C03649=1163.496,44.523,-49.145,-179.678,6.140,149.011
C03650=1163.500,44.274,-49.130,-179.680,6.139,149.011
C03651=1163.506,44.024,-49.115,-179.683,6.138,149.012
C03652=1163.511,43.775,-49.100,-179.686,6.137,149.012
C03653=1163.515,43.525,-49.084,-179.688,6.136,149.013
C03654=1163.521,43.275,-49.069,-179.691,6.135,149.014
C03655=1163.525,43.026,-49.054,-179.694,6.134,149.014
C03656=1163.531,42.777,-49.038,-179.696,6.133,149.015
C03657=1163.536,42.528,-49.023,-179.699,6.132,149.015
C03658=1163.540,42.278,-49.007,-179.701,6.131,149.016
C03659=1163.546,42.028,-48.992,-179.704,6.131,149.016
C03660=1163.551,41.779,-48.976,-179.707,6.129,149.017
C03661=1163.556,41.530,-48.961,-179.709,6.129,149.018
C03662=1163.561,41.280,-48.946,-179.711,6.128,149.018
C03663=1163.565,41.031,-48.930,-179.715,6.127,149.019
C03664=1163.571,40.781,-48.915,-179.717,6.126,149.019
C03665=1163.576,40.531,-48.900,-179.719,6.125,149.020
C03666=1163.581,40.282,-48.885,-179.722,6.124,149.020
C03667=1163.586,40.033,-48.869,-179.725,6.123,149.021
C03668=1163.591,39.784,-48.854,-179.727,6.122,149.021
C03669=1163.596,39.534,-48.839,-179.730,6.121,149.022
C03670=1163.601,39.284,-48.824,-179.732,6.120,149.022
C03671=1163.606,39.034,-48.808,-179.735,6.120,149.023
C03672=1163.611,38.785,-48.793,-179.737,6.119,149.024
C03673=1163.616,38.536,-48.778,-179.740,6.117,149.024
C03674=1163.621,38.286,-48.764,-179.742,6.117,149.025
C03675=1163.626,38.037,-48.748,-179.745,6.116,149.025
C03676=1163.632,37.787,-48.732,-179.748,6.114,149.026
C03677=1163.636,37.538,-48.717,-179.751,6.114,149.026
C03678=1163.642,37.288,-48.702,-179.753,6.113,149.027
C03679=1163.646,37.039,-48.687,-179.756,6.112,149.028
C03680=1163.652,36.789,-48.672,-179.758,6.111,149.028
C03681=1163.656,36.540,-48.657,-179.761,6.110,149.029
C03682=1163.661,36.290,-48.642,-179.763,6.110,149.029
C03683=1163.667,36.041,-48.627,-179.766,6.108,149.030
C03684=1163.671,35.792,-48.612,-179.768,6.107,149.030
C03685=1163.677,35.542,-48.597,-179.771,6.107,149.031
C03686=1163.682,35.293,-48.582,-179.774,6.105,149.031
C03687=1163.687,35.043,-48.566,-179.776,6.105,149.032
C03688=1163.692,34.794,-48.552,-179.779,6.104,149.033
C03689=1163.697,34.543,-48.536,-179.781,6.104,149.033
C03690=1163.702,34.294,-48.522,-179.784,6.102,149.034
C03691=1163.706,34.045,-48.507,-179.787,6.101,149.034
C03692=1163.712,33.795,-48.491,-179.789,6.101,149.035
C03693=1163.717,33.546,-48.477,-179.791,6.100,149.035
C03694=1163.722,33.296,-48.461,-179.795,6.099,149.036
C03695=1163.727,33.046,-48.447,-179.797,6.098,149.037
C03696=1163.732,32.797,-48.432,-179.799,6.097,149.037
C03697=1163.737,32.548,-48.416,-179.802,6.096,149.038
C03698=1163.742,32.298,-48.402,-179.805,6.095,149.038
C03699=1163.747,32.049,-48.387,-179.807,6.094,149.039
C03700=1163.752,31.799,-48.372,-179.810,6.094,149.040
C03701=1163.757,31.550,-48.357,-179.812,6.092,149.040
C03702=1163.763,31.300,-48.342,-179.815,6.092,149.041
C03703=1163.767,31.051,-48.327,-179.817,6.091,149.041
C03704=1163.772,30.801,-48.313,-179.820,6.091,149.042
C03705=1163.777,30.552,-48.298,-179.823,6.089,149.042
C03706=1163.783,30.302,-48.283,-179.825,6.088,149.043
C03707=1163.787,30.053,-48.268,-179.828,6.088,149.044
C03708=1163.792,29.803,-48.254,-179.830,6.087,149.044
C03709=1163.798,29.554,-48.238,-179.833,6.086,149.045
C03710=1163.803,29.304,-48.224,-179.835,6.085,149.045
C03711=1163.807,29.054,-48.210,-179.838,6.084,149.046
C03712=1163.813,28.805,-48.194,-179.840,6.084,149.046
C03713=1163.818,28.555,-48.180,-179.843,6.082,149.047
C03714=1163.823,28.287,-48.164,-179.846,6.082,149.048
C03715=1163.829,28.017,-48.148,-179.848,6.081,149.048
C03716=1163.834,27.749,-48.132,-179.851,6.080,149.049
C03717=1163.839,27.480,-48.117,-179.854,6.079,149.049
C03718=1163.844,27.230,-48.102,-179.856,6.078,149.050
C03719=1163.850,26.982,-48.087,-179.860,6.077,149.051
C03720=1163.855,26.732,-48.073,-179.862,6.076,149.051
C03721=1163.860,26.482,-48.059,-179.864,6.076,149.052
C03722=1163.865,26.233,-48.044,-179.866,6.075,149.052
C03723=1163.870,25.983,-48.029,-179.870,6.074,149.053
C03724=1163.875,25.733,-48.014,-179.872,6.073,149.054
C03725=1163.880,25.484,-47.999,-179.875,6.072,149.054
C03726=1163.885,25.234,-47.985,-179.877,6.072,149.055
C03727=1163.890,24.985,-47.971,-179.879,6.071,149.055
C03728=1163.895,24.735,-47.955,-179.883,6.070,149.056
C03729=1163.900,24.486,-47.941,-179.885,6.069,149.056
C03730=1163.905,24.236,-47.927,-179.887,6.069,149.057
C03731=1163.911,23.987,-47.913,-179.890,6.068,149.057
C03732=1163.915,23.738,-47.898,-179.893,6.066,149.058
C03733=1163.920,23.488,-47.884,-179.895,6.066,149.059
C03734=1163.925,23.238,-47.869,-179.898,6.065,149.059
C03735=1163.931,22.988,-47.854,-179.900,6.065,149.060
C03736=1163.936,22.739,-47.840,-179.902,6.064,149.060
C03737=1163.940,22.490,-47.825,-179.906,6.062,149.061
C03738=1163.945,22.240,-47.811,-179.908,6.062,149.061
C03739=1163.951,21.991,-47.797,-179.910,6.061,149.062
C03740=1163.956,21.741,-47.783,-179.913,6.060,149.063
C03741=1163.961,21.491,-47.768,-179.915,6.060,149.063
C03742=1163.966,21.242,-47.753,-179.918,6.058,149.064
C03743=1163.970,20.993,-47.739,-179.921,6.058,149.064
C03744=1163.976,20.743,-47.724,-179.923,6.057,149.065
C03745=1163.981,20.493,-47.710,-179.926,6.056,149.066
C03746=1163.987,20.244,-47.696,-179.928,6.056,149.066
C03747=1163.992,19.994,-47.682,-179.931,6.054,149.067
C03748=1163.997,19.744,-47.667,-179.934,6.054,149.067
C03749=1164.002,19.495,-47.653,-179.936,6.053,149.068
C03750=1164.006,19.246,-47.638,-179.938,6.053,149.069
C03751=1164.012,18.997,-47.624,-179.941,6.052,149.069
C03752=1164.017,18.747,-47.610,-179.943,6.051,149.070
C03753=1164.022,18.497,-47.596,-179.946,6.050,149.070
C03754=1164.027,18.248,-47.581,-179.949,6.049,149.071
C03755=1164.032,17.998,-47.567,-179.951,6.049,149.071
C03756=1164.037,17.749,-47.553,-179.953,6.048,149.072
C03757=1164.042,17.499,-47.539,-179.956,6.047,149.073
C03758=1164.047,17.249,-47.525,-179.959,6.046,149.073
C03759=1164.052,17.000,-47.510,-179.961,6.045,149.074
C03760=1164.057,16.750,-47.496,-179.964,6.044,149.074
C03761=1164.063,16.501,-47.482,-179.966,6.044,149.075
C03762=1164.067,16.251,-47.468,-179.968,6.043,149.075
C03763=1164.072,16.002,-47.454,-179.971,6.043,149.076
C03764=1164.077,15.752,-47.439,-179.974,6.041,149.077
C03765=1164.083,15.503,-47.426,-179.977,6.041,149.077
C03766=1164.088,15.253,-47.411,-179.979,6.040,149.078
C03767=1164.093,15.003,-47.397,-179.981,6.039,149.078
C03768=1164.098,14.754,-47.383,-179.984,6.039,149.079
C03769=1164.103,14.504,-47.370,-179.986,6.038,149.079
C03770=1164.108,14.255,-47.356,-179.989,6.037,149.080
C03771=1164.113,14.005,-47.342,-179.992,6.036,149.081
C03772=1164.118,13.756,-47.328,-179.994,6.035,149.081
C03773=1164.123,13.506,-47.313,-179.997,6.035,149.082
C03774=1164.128,13.257,-47.299,-179.999,6.034,149.082
C03775=1164.133,13.007,-47.285,179.998,6.034,149.083
C03776=1164.139,12.758,-47.271,179.996,6.033,149.084
C03777=1164.144,12.508,-47.257,179.993,6.032,149.084
C03778=1164.149,12.258,-47.243,179.991,6.031,149.085
C03779=1164.154,12.009,-47.230,179.988,6.030,149.085
C03780=1164.159,11.759,-47.215,179.985,6.030,149.086
C03781=1164.164,11.510,-47.201,179.983,6.029,149.087
C03782=1164.169,11.261,-47.187,179.981,6.028,149.087
C03783=1164.175,11.010,-47.174,179.978,6.028,149.088
C03784=1164.180,10.761,-47.159,179.976,6.027,149.088
C03785=1164.184,10.511,-47.146,179.973,6.026,149.089
C03786=1164.189,10.262,-47.132,179.970,6.025,149.089
C03787=1164.194,10.012,-47.118,179.968,6.025,149.090
C03788=1164.200,9.762,-47.104,179.966,6.024,149.091
C03789=1164.205,9.513,-47.090,179.963,6.023,149.091
C03790=1164.210,9.263,-47.076,179.961,6.022,149.092
C03791=1164.215,9.015,-47.062,179.958,6.022,149.092
C03792=1164.220,8.764,-47.049,179.956,6.021,149.093
C03793=1164.225,8.515,-47.035,179.953,6.020,149.094
C03794=1164.231,8.266,-47.021,179.950,6.019,149.094
C03795=1164.235,8.016,-47.008,179.948,6.019,149.095
C03796=1164.240,7.766,-46.993,179.945,6.018,149.095
C03797=1164.246,7.517,-46.980,179.943,6.017,149.096
C03798=1164.251,7.267,-46.966,179.940,6.017,149.097
C03799=1164.256,7.018,-46.953,179.938,6.016,149.097
C03800=1164.261,6.768,-46.938,179.936,6.016,149.098
C03801=1164.266,6.518,-46.925,179.933,6.014,149.098
C03802=1164.272,6.269,-46.911,179.930,6.013,149.099
C03803=1164.276,6.019,-46.897,179.927,6.013,149.100
C03804=1164.281,5.769,-46.884,179.925,6.012,149.100
C03805=1164.287,5.520,-46.870,179.923,6.012,149.101
C03806=1164.291,5.271,-46.856,179.920,6.011,149.101
C03807=1164.297,5.021,-46.843,179.918,6.010,149.102
C03808=1164.302,4.771,-46.829,179.916,6.010,149.102
C03809=1164.307,4.522,-46.815,179.913,6.009,149.103
C03810=1164.312,4.272,-46.802,179.910,6.009,149.104
C03811=1164.317,4.022,-46.788,179.908,6.007,149.104
C03812=1164.322,3.773,-46.774,179.905,6.007,149.105
C03813=1164.327,3.524,-46.761,179.903,6.006,149.105
C03814=1164.333,3.274,-46.747,179.900,6.005,149.106
C03815=1164.337,3.024,-46.733,179.898,6.005,149.106
C03816=1164.343,2.775,-46.721,179.895,6.004,149.107
C03817=1164.348,2.525,-46.706,179.893,6.004,149.108
C03818=1164.353,2.255,-46.692,179.890,6.003,149.108
C03819=1164.359,1.987,-46.678,179.887,6.002,149.109
C03820=1164.364,1.717,-46.663,179.885,6.001,149.110
C03821=1164.369,1.448,-46.648,179.882,6.001,149.110
C03822=1164.375,1.198,-46.635,179.880,6.000,149.111
C03823=1164.380,0.949,-46.621,179.877,5.999,149.112
C03824=1164.385,0.699,-46.608,179.875,5.998,149.112
C03825=1164.390,0.449,-46.595,179.872,5.998,149.113
C03826=1164.395,0.200,-46.581,179.870,5.998,149.113
C03827=1164.401,-0.050,-46.567,179.867,5.997,149.114
C03828=1164.406,-0.299,-46.554,179.864,5.996,149.115
C03829=1164.411,-0.549,-46.541,179.862,5.995,149.115
C03830=1164.416,-0.798,-46.528,179.859,5.994,149.116
C03831=1164.421,-1.048,-46.514,179.857,5.993,149.116
C03832=1164.426,-1.297,-46.501,179.855,5.993,149.117
C03833=1164.431,-1.547,-46.487,179.852,5.993,149.117
C03834=1164.436,-1.796,-46.474,179.850,5.992,149.118
C03835=1164.441,-2.047,-46.461,179.847,5.991,149.119
C03836=1164.446,-2.295,-46.447,179.845,5.990,149.119
C03837=1164.451,-2.546,-46.434,179.842,5.990,149.120
C03838=1164.457,-2.795,-46.421,179.840,5.989,149.120
C03839=1164.462,-3.045,-46.407,179.837,5.989,149.121
C03840=1164.467,-3.294,-46.394,179.835,5.988,149.122
C03841=1164.472,-3.544,-46.381,179.833,5.987,149.122
C03842=1164.477,-3.793,-46.367,179.830,5.987,149.123
C03843=1164.483,-4.043,-46.354,179.828,5.986,149.123
C03844=1164.487,-4.293,-46.341,179.825,5.986,149.124
C03845=1164.493,-4.542,-46.328,179.822,5.984,149.125
C03846=1164.497,-4.792,-46.314,179.820,5.984,149.125
C03847=1164.503,-5.041,-46.301,179.817,5.983,149.126
C03848=1164.508,-5.292,-46.288,179.815,5.982,149.126
C03849=1164.513,-5.541,-46.275,179.812,5.982,149.127
C03850=1164.518,-5.790,-46.262,179.810,5.981,149.127
C03851=1164.524,-6.040,-46.248,179.807,5.981,149.128
C03852=1164.529,-6.289,-46.236,179.805,5.980,149.129
C03853=1164.533,-6.539,-46.223,179.802,5.979,149.129
C03854=1164.539,-6.789,-46.209,179.800,5.979,149.130
C03855=1164.544,-7.038,-46.196,179.798,5.978,149.130
C03856=1164.549,-7.288,-46.183,179.795,5.978,149.131
C03857=1164.554,-7.537,-46.170,179.793,5.977,149.132
C03858=1164.559,-7.787,-46.157,179.790,5.976,149.132
C03859=1164.565,-8.037,-46.144,179.788,5.976,149.133
C03860=1164.569,-8.286,-46.130,179.785,5.975,149.133
C03861=1164.575,-8.536,-46.117,179.783,5.975,149.134
C03862=1164.580,-8.785,-46.104,179.780,5.974,149.135
C03863=1164.585,-9.035,-46.092,179.778,5.973,149.135
C03864=1164.590,-9.285,-46.078,179.776,5.973,149.136
C03865=1164.595,-9.534,-46.065,179.773,5.972,149.136
C03866=1164.600,-9.784,-46.053,179.770,5.972,149.137
C03867=1164.606,-10.034,-46.039,179.768,5.971,149.138
C03868=1164.611,-10.283,-46.026,179.766,5.970,149.138
C03869=1164.615,-10.533,-46.013,179.763,5.970,149.139
C03870=1164.621,-10.782,-46.000,179.761,5.969,149.139
C03871=1164.626,-11.032,-45.987,179.758,5.969,149.140
C03872=1164.631,-11.282,-45.974,179.756,5.968,149.141
C03873=1164.636,-11.531,-45.961,179.753,5.967,149.141
C03874=1164.642,-11.781,-45.948,179.751,5.967,149.142
C03875=1164.646,-12.031,-45.936,179.748,5.966,149.142
C03876=1164.651,-12.280,-45.923,179.746,5.965,149.143
C03877=1164.657,-12.530,-45.910,179.744,5.965,149.144
C03878=1164.662,-12.779,-45.897,179.741,5.964,149.144
C03879=1164.667,-13.029,-45.884,179.739,5.964,149.145
C03880=1164.673,-13.279,-45.871,179.736,5.963,149.145
C03881=1164.678,-13.528,-45.858,179.734,5.962,149.146
C03882=1164.682,-13.778,-45.845,179.731,5.962,149.147
C03883=1164.687,-14.027,-45.833,179.729,5.961,149.147
C03884=1164.693,-14.277,-45.820,179.726,5.961,149.148
C03885=1164.698,-14.527,-45.807,179.724,5.960,149.148
C03886=1164.703,-14.776,-45.794,179.722,5.959,149.149
C03887=1164.708,-15.026,-45.781,179.719,5.959,149.150
C03888=1164.713,-15.275,-45.769,179.717,5.958,149.150
C03889=1164.719,-15.526,-45.756,179.714,5.958,149.151
C03890=1164.724,-15.775,-45.743,179.711,5.957,149.151
C03891=1164.729,-16.024,-45.731,179.709,5.956,149.152
C03892=1164.734,-16.274,-45.718,179.707,5.956,149.153
C03893=1164.739,-16.524,-45.705,179.704,5.955,149.153
C03894=1164.744,-16.773,-45.692,179.702,5.955,149.154
C03895=1164.750,-17.023,-45.679,179.700,5.954,149.154
C03896=1164.755,-17.272,-45.667,179.697,5.953,149.155
C03897=1164.759,-17.523,-45.655,179.694,5.953,149.156
C03898=1164.765,-17.772,-45.642,179.692,5.952,149.156
C03899=1164.770,-18.021,-45.629,179.689,5.952,149.157
C03900=1164.776,-18.271,-45.616,179.687,5.951,149.157
C03901=1164.781,-18.520,-45.604,179.685,5.951,149.158
C03902=1164.785,-18.770,-45.591,179.682,5.950,149.158
C03903=1164.791,-19.020,-45.579,179.680,5.949,149.159
C03904=1164.796,-19.270,-45.566,179.677,5.949,149.160
C03905=1164.801,-19.519,-45.554,179.675,5.948,149.160
C03906=1164.806,-19.768,-45.541,179.672,5.948,149.161
C03907=1164.811,-20.019,-45.527,179.670,5.947,149.161
C03908=1164.817,-20.268,-45.515,179.667,5.946,149.162
C03909=1164.822,-20.518,-45.503,179.665,5.946,149.163
C03910=1164.827,-20.767,-45.490,179.663,5.946,149.163
C03911=1164.832,-21.017,-45.478,179.660,5.945,149.164
C03912=1164.838,-21.266,-45.466,179.658,5.945,149.165
C03913=1164.842,-21.516,-45.453,179.656,5.944,149.165
C03914=1164.847,-21.766,-45.440,179.653,5.943,149.166
C03915=1164.853,-22.016,-45.428,179.651,5.943,149.166
C03916=1164.858,-22.265,-45.416,179.648,5.943,149.167
C03917=1164.863,-22.514,-45.403,179.646,5.942,149.168
C03918=1164.868,-22.764,-45.391,179.643,5.941,149.168
C03919=1164.874,-23.015,-45.378,179.641,5.940,149.169
C03920=1164.879,-23.264,-45.365,179.638,5.940,149.169
C03921=1164.884,-23.514,-45.353,179.636,5.939,149.170
C03922=1164.890,-23.783,-45.340,179.634,5.939,149.171
C03923=1164.895,-24.053,-45.327,179.631,5.938,149.171
C03924=1164.901,-24.323,-45.313,179.628,5.938,149.172
C03925=1164.906,-24.592,-45.299,179.626,5.937,149.173
C03926=1164.911,-24.843,-45.287,179.623,5.937,149.173
C03927=1164.916,-25.092,-45.274,179.621,5.936,149.174
C03928=1164.922,-25.342,-45.263,179.619,5.935,149.174
C03929=1164.927,-25.591,-45.250,179.616,5.935,149.175
C03930=1164.932,-25.841,-45.237,179.614,5.934,149.175
C03931=1164.937,-26.091,-45.226,179.611,5.934,149.176
C03932=1164.943,-26.340,-45.213,179.608,5.933,149.177
C03933=1164.948,-26.590,-45.201,179.606,5.932,149.177
C03934=1164.953,-26.839,-45.188,179.604,5.932,149.178
C03935=1164.959,-27.089,-45.177,179.601,5.931,149.178
C03936=1164.962,-27.339,-45.164,179.599,5.932,149.179
C03937=1164.968,-27.589,-45.152,179.597,5.931,149.180
C03938=1164.973,-27.838,-45.140,179.594,5.930,149.180
C03939=1164.978,-28.088,-45.128,179.592,5.930,149.181
C03940=1164.983,-28.337,-45.115,179.590,5.929,149.182
C03941=1164.989,-28.587,-45.103,179.587,5.929,149.182
C03942=1164.994,-28.837,-45.091,179.585,5.928,149.183
C03943=1164.999,-29.087,-45.079,179.582,5.927,149.183
C03944=1165.005,-29.336,-45.066,179.580,5.927,149.184
C03945=1165.010,-29.586,-45.054,179.577,5.926,149.185
C03946=1165.015,-29.835,-45.042,179.575,5.926,149.185
C03947=1165.020,-30.085,-45.030,179.572,5.925,149.186
C03948=1165.025,-30.334,-45.018,179.570,5.925,149.186
C03949=1165.030,-30.584,-45.006,179.568,5.925,149.187
C03950=1165.035,-30.833,-44.993,179.566,5.924,149.188
C03951=1165.041,-31.083,-44.981,179.563,5.923,149.188
C03952=1165.046,-31.333,-44.970,179.561,5.923,149.189
C03953=1165.051,-31.583,-44.957,179.558,5.922,149.189
C03954=1165.056,-31.832,-44.946,179.556,5.922,149.190
C03955=1165.061,-32.082,-44.933,179.553,5.921,149.191
C03956=1165.067,-32.331,-44.921,179.551,5.920,149.191
C03957=1165.072,-32.581,-44.909,179.549,5.921,149.192
C03958=1165.077,-32.831,-44.897,179.547,5.920,149.192
C03959=1165.083,-33.081,-44.885,179.544,5.920,149.193
C03960=1165.087,-33.330,-44.874,179.541,5.919,149.194
C03961=1165.092,-33.580,-44.861,179.539,5.918,149.194
C03962=1165.098,-33.830,-44.849,179.537,5.918,149.195
C03963=1165.103,-34.079,-44.837,179.534,5.917,149.195
C03964=1165.108,-34.329,-44.825,179.532,5.917,149.196
C03965=1165.113,-34.578,-44.813,179.530,5.916,149.196
C03966=1165.119,-34.828,-44.801,179.528,5.916,149.197
C03967=1165.124,-35.078,-44.789,179.525,5.916,149.198
C03968=1165.129,-35.328,-44.777,179.523,5.915,149.198
C03969=1165.135,-35.578,-44.765,179.520,5.915,149.199
C03970=1165.139,-35.827,-44.754,179.518,5.914,149.200
C03971=1165.144,-36.076,-44.741,179.515,5.913,149.200
C03972=1165.150,-36.326,-44.729,179.513,5.913,149.201
C03973=1165.155,-36.576,-44.717,179.510,5.912,149.201
C03974=1165.160,-36.826,-44.706,179.509,5.912,149.202
C03975=1165.165,-37.075,-44.693,179.506,5.912,149.203
C03976=1165.170,-37.325,-44.682,179.503,5.911,149.203
C03977=1165.175,-37.575,-44.670,179.501,5.910,149.204
C03978=1165.181,-37.825,-44.658,179.499,5.910,149.204
C03979=1165.186,-38.073,-44.646,179.496,5.909,149.205
C03980=1165.192,-38.323,-44.634,179.494,5.909,149.206
C03981=1165.196,-38.573,-44.623,179.492,5.908,149.206
C03982=1165.202,-38.823,-44.611,179.489,5.908,149.207
C03983=1165.207,-39.073,-44.599,179.487,5.908,149.208
C03984=1165.212,-39.322,-44.588,179.485,5.907,149.208
C03985=1165.217,-39.572,-44.575,179.482,5.907,149.209
C03986=1165.223,-39.822,-44.563,179.480,5.906,149.209
C03987=1165.227,-40.071,-44.552,179.477,5.905,149.210
C03988=1165.233,-40.321,-44.540,179.475,5.905,149.210
C03989=1165.239,-40.571,-44.529,179.473,5.905,149.211
C03990=1165.243,-40.820,-44.517,179.471,5.904,149.211
C03991=1165.249,-41.070,-44.506,179.468,5.904,149.212
C03992=1165.254,-41.320,-44.494,179.465,5.903,149.213
C03993=1165.259,-41.569,-44.482,179.463,5.903,149.213
C03994=1165.264,-41.819,-44.470,179.460,5.902,149.214
C03995=1165.269,-42.069,-44.458,179.459,5.902,149.215
C03996=1165.274,-42.319,-44.447,179.456,5.902,149.215
C03997=1165.280,-42.568,-44.435,179.454,5.901,149.216
C03998=1165.285,-42.817,-44.424,179.451,5.901,149.216
C03999=1165.290,-43.067,-44.412,179.449,5.900,149.217
C04000=1165.296,-43.317,-44.400,179.447,5.899,149.218
C04001=1165.300,-43.567,-44.389,179.444,5.899,149.218
C04002=1165.306,-43.817,-44.377,179.442,5.899,149.219
C04003=1165.311,-44.066,-44.366,179.440,5.898,149.219
C04004=1165.317,-44.316,-44.354,179.437,5.898,149.220
C04005=1165.321,-44.565,-44.343,179.435,5.897,149.221
C04006=1165.327,-44.815,-44.331,179.433,5.896,149.221
C04007=1165.332,-45.065,-44.319,179.430,5.896,149.222
C04008=1165.337,-45.315,-44.308,179.428,5.896,149.222
C04009=1165.343,-45.564,-44.296,179.426,5.896,149.223
C04010=1165.348,-45.814,-44.285,179.423,5.895,149.224
C04011=1165.353,-46.064,-44.273,179.421,5.894,149.224
C04012=1165.358,-46.313,-44.262,179.418,5.894,149.225
C04013=1165.363,-46.563,-44.250,179.417,5.894,149.225
C04014=1165.368,-46.812,-44.239,179.414,5.894,149.226
C04015=1165.374,-47.062,-44.227,179.412,5.893,149.227
C04016=1165.379,-47.312,-44.216,179.409,5.892,149.227
C04017=1165.384,-47.562,-44.204,179.407,5.892,149.228
C04018=1165.389,-47.812,-44.193,179.404,5.891,149.228
C04019=1165.395,-48.061,-44.182,179.402,5.892,149.229
C04020=1165.400,-48.311,-44.170,179.400,5.891,149.230
C04021=1165.405,-48.561,-44.159,179.397,5.890,149.230
C04022=1165.410,-48.810,-44.147,179.395,5.889,149.231
C04023=1165.416,-49.059,-44.136,179.392,5.889,149.231
C04024=1165.421,-49.309,-44.125,179.391,5.889,149.232
C04025=1165.426,-49.559,-44.113,179.388,5.889,149.233
C04026=1165.432,-49.829,-44.101,179.385,5.888,149.233
C04027=1165.437,-50.100,-44.089,179.383,5.887,149.234
C04028=1165.442,-50.370,-44.076,179.381,5.887,149.235
C04029=1165.449,-50.641,-44.064,179.378,5.887,149.235
C04030=1165.454,-50.891,-44.052,179.376,5.886,149.236
C04031=1165.459,-51.141,-44.042,179.373,5.885,149.236
C04032=1165.464,-51.390,-44.030,179.371,5.885,149.237
C04033=1165.470,-51.640,-44.019,179.369,5.885,149.238
C04034=1165.474,-51.889,-44.008,179.366,5.885,149.238
C04035=1165.480,-52.139,-43.996,179.364,5.884,149.239
C04036=1165.485,-52.389,-43.986,179.361,5.883,149.240
C04037=1165.490,-52.638,-43.974,179.360,5.883,149.240
C04038=1165.496,-52.888,-43.962,179.357,5.883,149.241
C04039=1165.500,-53.138,-43.951,179.355,5.882,149.241
C04040=1165.507,-53.388,-43.940,179.352,5.882,149.242
C04041=1165.511,-53.637,-43.929,179.350,5.881,149.242
C04042=1165.516,-53.887,-43.918,179.348,5.881,149.243
C04043=1165.522,-54.136,-43.906,179.346,5.881,149.244
C04044=1165.527,-54.387,-43.896,179.343,5.880,149.244
C04045=1165.532,-54.636,-43.884,179.340,5.880,149.245
C04046=1165.538,-54.885,-43.873,179.338,5.879,149.245
C04047=1165.543,-55.136,-43.862,179.336,5.879,149.246
C04048=1165.547,-55.385,-43.851,179.334,5.879,149.247
C04049=1165.553,-55.635,-43.839,179.331,5.878,149.247
C04050=1165.558,-55.885,-43.829,179.329,5.877,149.248
C04051=1165.563,-56.134,-43.818,179.327,5.878,149.248
C04052=1165.569,-56.384,-43.806,179.325,5.877,149.249
C04053=1165.574,-56.634,-43.795,179.322,5.877,149.250
C04054=1165.579,-56.883,-43.784,179.320,5.876,149.250
C04055=1165.584,-57.132,-43.773,179.317,5.875,149.251
C04056=1165.590,-57.383,-43.762,179.316,5.875,149.251
C04057=1165.595,-57.633,-43.751,179.313,5.875,149.252
C04058=1165.600,-57.882,-43.741,179.311,5.874,149.252
C04059=1165.606,-58.132,-43.729,179.308,5.874,149.253
C04060=1165.610,-58.382,-43.717,179.306,5.874,149.254
C04061=1165.616,-58.631,-43.707,179.304,5.873,149.254
C04062=1165.621,-58.881,-43.696,179.301,5.873,149.255
C04063=1165.627,-59.131,-43.685,179.299,5.872,149.256
C04064=1165.632,-59.380,-43.674,179.297,5.872,149.256
C04065=1165.637,-59.631,-43.663,179.295,5.872,149.257
C04066=1165.642,-59.880,-43.652,179.292,5.871,149.257
C04067=1165.647,-60.129,-43.641,179.290,5.870,149.258
C04068=1165.652,-60.380,-43.630,179.288,5.871,149.259
C04069=1165.658,-60.629,-43.619,179.286,5.870,149.259
C04070=1165.663,-60.879,-43.608,179.283,5.870,149.260
C04071=1165.668,-61.128,-43.597,179.281,5.869,149.260
C04072=1165.674,-61.378,-43.586,179.279,5.869,149.261
C04073=1165.679,-61.627,-43.575,179.277,5.868,149.261
C04074=1165.684,-61.878,-43.565,179.274,5.868,149.262
C04075=1165.689,-62.127,-43.553,179.272,5.867,149.263
C04076=1165.694,-62.377,-43.543,179.270,5.868,149.263
C04077=1165.699,-62.626,-43.532,179.267,5.867,149.264
C04078=1165.705,-62.876,-43.521,179.265,5.866,149.265
C04079=1165.710,-63.126,-43.511,179.263,5.866,149.265
C04080=1165.716,-63.375,-43.500,179.261,5.866,149.266
C04081=1165.721,-63.626,-43.489,179.258,5.865,149.266
C04082=1165.725,-63.875,-43.478,179.256,5.865,149.267
C04083=1165.731,-64.125,-43.468,179.253,5.864,149.268
C04084=1165.736,-64.375,-43.456,179.251,5.864,149.268
C04085=1165.742,-64.624,-43.446,179.249,5.864,149.269
C04086=1165.747,-64.874,-43.435,179.247,5.863,149.269
C04087=1165.752,-65.123,-43.424,179.244,5.863,149.270
C04088=1165.757,-65.374,-43.413,179.242,5.863,149.270
C04089=1165.762,-65.623,-43.403,179.240,5.863,149.271
C04090=1165.767,-65.873,-43.392,179.237,5.862,149.272
C04091=1165.773,-66.122,-43.382,179.235,5.862,149.272
C04092=1165.778,-66.372,-43.370,179.233,5.861,149.273
C04093=1165.784,-66.622,-43.360,179.231,5.861,149.274
C04094=1165.789,-66.872,-43.349,179.228,5.860,149.274
C04095=1165.794,-67.121,-43.338,179.226,5.861,149.275
C04096=1165.799,-67.371,-43.328,179.224,5.860,149.275
C04097=1165.805,-67.621,-43.317,179.221,5.859,149.276
C04098=1165.810,-67.870,-43.306,179.219,5.859,149.276
C04099=1165.815,-68.120,-43.296,179.217,5.859,149.277
C04100=1165.820,-68.370,-43.285,179.215,5.858,149.278
C04101=1165.826,-68.619,-43.274,179.212,5.858,149.278
C04102=1165.831,-68.869,-43.264,179.211,5.858,149.279
C04103=1165.836,-69.119,-43.254,179.208,5.857,149.279
C04104=1165.841,-69.369,-43.243,179.206,5.857,149.280
C04105=1165.846,-69.618,-43.232,179.203,5.856,149.281
C04106=1165.851,-69.868,-43.222,179.202,5.856,149.281
C04107=1165.857,-70.118,-43.211,179.199,5.856,149.282
C04108=1165.863,-70.368,-43.200,179.197,5.855,149.282
C04109=1165.868,-70.617,-43.189,179.195,5.855,149.283
C04110=1165.873,-70.868,-43.179,179.192,5.855,149.284
C04111=1165.879,-71.117,-43.168,179.190,5.854,149.284
C04112=1165.884,-71.367,-43.158,179.188,5.853,149.285
C04113=1165.889,-71.616,-43.147,179.186,5.854,149.285
C04114=1165.895,-71.866,-43.137,179.183,5.853,149.286
C04115=1165.900,-72.116,-43.126,179.181,5.853,149.287
C04116=1165.905,-72.366,-43.116,179.179,5.853,149.287
C04117=1165.910,-72.616,-43.105,179.176,5.852,149.288
C04118=1165.916,-72.865,-43.095,179.174,5.851,149.288
C04119=1165.920,-73.114,-43.085,179.172,5.852,149.289
C04120=1165.925,-73.364,-43.074,179.170,5.851,149.289
C04121=1165.931,-73.614,-43.064,179.167,5.851,149.290
C04122=1165.936,-73.864,-43.053,179.165,5.850,149.291
C04123=1165.941,-74.114,-43.043,179.163,5.850,149.291
C04124=1165.947,-74.363,-43.033,179.161,5.849,149.292
C04125=1165.952,-74.613,-43.022,179.158,5.849,149.293
C04126=1165.957,-74.862,-43.012,179.157,5.849,149.293
C04127=1165.962,-75.113,-43.001,179.154,5.849,149.294
C04128=1165.968,-75.362,-42.991,179.152,5.848,149.294
C04129=1165.974,-75.612,-42.981,179.150,5.848,149.295
C04130=1165.979,-75.883,-42.970,179.147,5.848,149.295
C04131=1165.985,-76.155,-42.958,179.145,5.847,149.296
C04132=1165.991,-76.425,-42.947,179.142,5.847,149.297
C04133=1165.996,-76.697,-42.936,179.140,5.846,149.297
C04134=1166.002,-76.946,-42.926,179.138,5.846,149.298
C04135=1166.007,-77.197,-42.915,179.136,5.846,149.299
C04136=1166.013,-77.446,-42.905,179.133,5.845,149.299
C04137=1166.018,-77.696,-42.895,179.131,5.845,149.300
C04138=1166.023,-77.945,-42.883,179.129,5.845,149.300
C04139=1166.028,-78.194,-42.874,179.126,5.844,149.301
C04140=1166.033,-78.444,-42.864,179.124,5.844,149.302
C04141=1166.038,-78.694,-42.853,179.122,5.844,149.302
C04142=1166.044,-78.944,-42.843,179.120,5.843,149.303
C04143=1166.050,-79.193,-42.833,179.118,5.843,149.303
C04144=1166.055,-79.444,-42.822,179.115,5.843,149.304
C04145=1166.059,-79.693,-42.812,179.113,5.842,149.304
C04146=1166.065,-79.943,-42.803,179.111,5.842,149.305
C04147=1166.070,-80.193,-42.792,179.109,5.842,149.306
C04148=1166.076,-80.443,-42.782,179.107,5.841,149.306
C04149=1166.081,-80.692,-42.772,179.105,5.841,149.307
C04150=1166.086,-80.943,-42.761,179.102,5.841,149.307
C04151=1166.091,-81.192,-42.752,179.100,5.840,149.308
C04152=1166.097,-81.441,-42.742,179.098,5.840,149.309
C04153=1166.102,-81.692,-42.731,179.095,5.840,149.309
C04154=1166.108,-81.941,-42.721,179.093,5.839,149.310
C04155=1166.113,-82.191,-42.711,179.091,5.839,149.310
C04156=1166.117,-82.441,-42.701,179.089,5.839,149.311
C04157=1166.123,-82.690,-42.690,179.086,5.838,149.312
C04158=1166.129,-82.940,-42.680,179.085,5.838,149.312
C04159=1166.134,-83.190,-42.671,179.082,5.838,149.313
C04160=1166.139,-83.440,-42.661,179.080,5.837,149.313
C04161=1166.144,-83.689,-42.651,179.078,5.837,149.314
C04162=1166.150,-83.939,-42.640,179.076,5.837,149.314
C04163=1166.155,-84.189,-42.630,179.073,5.836,149.315
C04164=1166.160,-84.438,-42.620,179.071,5.836,149.316
C04165=1166.165,-84.688,-42.610,179.069,5.836,149.316
C04166=1166.171,-84.938,-42.600,179.066,5.835,149.317
C04167=1166.176,-85.188,-42.590,179.065,5.835,149.317
C04168=1166.181,-85.438,-42.580,179.062,5.835,149.318
C04169=1166.187,-85.687,-42.570,179.060,5.834,149.319
C04170=1166.192,-85.937,-42.560,179.058,5.834,149.319
C04171=1166.197,-86.187,-42.550,179.056,5.834,149.320
C04172=1166.203,-86.437,-42.540,179.054,5.834,149.320
C04173=1166.208,-86.686,-42.530,179.051,5.833,149.321
C04174=1166.213,-86.935,-42.521,179.049,5.832,149.321
C04175=1166.218,-87.186,-42.510,179.047,5.833,149.322
C04176=1166.224,-87.436,-42.500,179.045,5.832,149.323
C04177=1166.229,-87.685,-42.491,179.042,5.832,149.323
C04178=1166.234,-87.935,-42.481,179.041,5.832,149.324
C04179=1166.240,-88.184,-42.470,179.038,5.831,149.325
C04180=1166.245,-88.435,-42.461,179.036,5.831,149.325
C04181=1166.250,-88.684,-42.451,179.034,5.831,149.325
C04182=1166.256,-88.934,-42.441,179.032,5.830,149.326
C04183=1166.261,-89.183,-42.431,179.030,5.830,149.327
C04184=1166.266,-89.434,-42.421,179.027,5.830,149.327
C04185=1166.271,-89.683,-42.412,179.025,5.829,149.328
C04186=1166.276,-89.933,-42.401,179.023,5.829,149.329
C04187=1166.282,-90.183,-42.392,179.021,5.829,149.329
C04188=1166.287,-90.432,-42.382,179.019,5.828,149.330
C04189=1166.293,-90.682,-42.372,179.017,5.828,149.330
C04190=1166.298,-90.933,-42.362,179.014,5.828,149.331
C04191=1166.303,-91.182,-42.353,179.012,5.828,149.331
C04192=1166.308,-91.431,-42.342,179.010,5.827,149.332
C04193=1166.314,-91.681,-42.334,179.007,5.827,149.333
C04194=1166.319,-91.931,-42.323,179.006,5.827,149.333
C04195=1166.325,-92.180,-42.313,179.004,5.826,149.334
C04196=1166.329,-92.431,-42.304,179.001,5.826,149.334
C04197=1166.335,-92.680,-42.294,178.999,5.826,149.335
C04198=1166.340,-92.930,-42.284,178.997,5.825,149.336
C04199=1166.346,-93.180,-42.275,178.995,5.825,149.336
C04200=1166.351,-93.429,-42.265,178.992,5.825,149.337
C04201=1166.357,-93.679,-42.255,178.990,5.824,149.337
C04202=1166.361,-93.929,-42.245,178.989,5.824,149.338
C04203=1166.366,-94.179,-42.235,178.986,5.824,149.338
C04204=1166.372,-94.429,-42.226,178.984,5.824,149.339
C04205=1166.377,-94.678,-42.216,178.982,5.823,149.340
C04206=1166.383,-94.928,-42.207,178.979,5.823,149.340
C04207=1166.388,-95.177,-42.197,178.977,5.823,149.341
C04208=1166.394,-95.428,-42.188,178.975,5.822,149.341
C04209=1166.399,-95.677,-42.178,178.974,5.822,149.342
C04210=1166.404,-95.928,-42.168,178.971,5.822,149.342
C04211=1166.409,-96.177,-42.158,178.969,5.821,149.343
C04212=1166.414,-96.426,-42.148,178.967,5.822,149.344
C04213=1166.420,-96.676,-42.139,178.964,5.821,149.344
C04214=1166.425,-96.926,-42.129,178.963,5.821,149.345
C04215=1166.430,-97.176,-42.120,178.960,5.820,149.345
C04216=1166.436,-97.425,-42.110,178.958,5.820,149.346
C04217=1166.441,-97.675,-42.101,178.956,5.820,149.347
C04218=1166.447,-97.925,-42.092,178.954,5.819,149.347
C04219=1166.452,-98.174,-42.082,178.952,5.819,149.347
C04220=1166.458,-98.425,-42.073,178.949,5.819,149.348
C04221=1166.463,-98.674,-42.063,178.947,5.818,149.349
C04222=1166.468,-98.925,-42.053,178.945,5.819,149.349
C04223=1166.473,-99.174,-42.043,178.943,5.818,149.350
C04224=1166.478,-99.424,-42.035,178.941,5.818,149.350
C04225=1166.484,-99.673,-42.024,178.939,5.817,149.351
C04226=1166.489,-99.923,-42.015,178.937,5.817,149.352
C04227=1166.494,-100.173,-42.005,178.934,5.817,149.352
C04228=1166.500,-100.423,-41.996,178.932,5.816,149.353
C04229=1166.505,-100.673,-41.987,178.931,5.816,149.353
C04230=1166.510,-100.922,-41.977,178.928,5.816,149.354
C04231=1166.515,-101.172,-41.968,178.926,5.816,149.354
C04232=1166.521,-101.421,-41.958,178.924,5.816,149.355
C04233=1166.526,-101.671,-41.949,178.922,5.815,149.356
C04234=1166.532,-101.943,-41.939,178.919,5.815,149.356
C04235=1166.538,-102.215,-41.928,178.917,5.814,149.357
C04236=1166.543,-102.487,-41.918,178.915,5.814,149.358
C04237=1166.550,-102.759,-41.908,178.913,5.814,149.358
C04238=1166.555,-103.008,-41.899,178.910,5.814,149.359
C04239=1166.561,-103.259,-41.890,178.908,5.813,149.359
C04240=1166.565,-103.508,-41.880,178.906,5.813,149.360
C04241=1166.571,-103.758,-41.871,178.904,5.813,149.360
C04242=1166.577,-104.008,-41.862,178.902,5.813,149.361
C04243=1166.581,-104.257,-41.852,178.900,5.812,149.362
C04244=1166.587,-104.507,-41.843,178.898,5.812,149.362
C04245=1166.592,-104.757,-41.834,178.896,5.812,149.363
C04246=1166.597,-105.006,-41.824,178.893,5.811,149.363
C04247=1166.602,-105.256,-41.815,178.892,5.811,149.364
C04248=1166.608,-105.506,-41.806,178.889,5.811,149.365
C04249=1166.614,-105.756,-41.797,178.887,5.811,149.365
C04250=1166.618,-106.005,-41.787,178.885,5.810,149.366
C04251=1166.624,-106.256,-41.778,178.883,5.810,149.366
C04252=1166.629,-106.505,-41.769,178.881,5.810,149.367
C04253=1166.635,-106.755,-41.760,178.879,5.809,149.367
C04254=1166.640,-107.005,-41.750,178.877,5.809,149.368
C04255=1166.645,-107.255,-41.741,178.874,5.809,149.368
C04256=1166.651,-107.504,-41.732,178.873,5.809,149.369
C04257=1166.656,-107.754,-41.723,178.870,5.808,149.370
C04258=1166.661,-108.004,-41.713,178.868,5.808,149.370
C04259=1166.667,-108.254,-41.704,178.866,5.808,149.371
C04260=1166.672,-108.504,-41.695,178.864,5.808,149.371
C04261=1166.677,-108.753,-41.686,178.862,5.807,149.372
C04262=1166.683,-109.004,-41.677,178.859,5.807,149.372
C04263=1166.688,-109.253,-41.667,178.858,5.807,149.373
C04264=1166.693,-109.503,-41.658,178.855,5.806,149.373
C04265=1166.698,-109.753,-41.649,178.853,5.806,149.374
C04266=1166.704,-110.003,-41.640,178.851,5.806,149.375
C04267=1166.709,-110.253,-41.631,178.850,5.806,149.375
C04268=1166.714,-110.502,-41.622,178.847,5.805,149.376
C04269=1166.720,-110.751,-41.613,178.845,5.805,149.376
C04270=1166.726,-111.001,-41.603,178.843,5.805,149.377
C04271=1166.731,-111.251,-41.594,178.841,5.805,149.378
C04272=1166.736,-111.501,-41.585,178.839,5.804,149.378
C04273=1166.741,-111.751,-41.576,178.837,5.803,149.379
C04274=1166.746,-112.000,-41.568,178.835,5.804,149.379
C04275=1166.752,-112.251,-41.558,178.832,5.803,149.380
C04276=1166.757,-112.501,-41.549,178.830,5.804,149.380
C04277=1166.762,-112.750,-41.540,178.828,5.803,149.381
C04278=1166.767,-113.000,-41.531,178.827,5.803,149.381
C04279=1166.773,-113.249,-41.522,178.824,5.802,149.382
C04280=1166.779,-113.499,-41.513,178.822,5.802,149.383
C04281=1166.784,-113.749,-41.504,178.820,5.802,149.383
C04282=1166.789,-113.999,-41.495,178.818,5.802,149.384
C04283=1166.794,-114.248,-41.486,178.816,5.801,149.384
C04284=1166.800,-114.498,-41.477,178.814,5.801,149.385
C04285=1166.805,-114.748,-41.468,178.812,5.801,149.385
C04286=1166.811,-114.998,-41.459,178.810,5.801,149.386
C04287=1166.816,-115.247,-41.450,178.808,5.800,149.386
C04288=1166.822,-115.497,-41.441,178.806,5.800,149.387
C04289=1166.827,-115.747,-41.432,178.803,5.800,149.388
C04290=1166.832,-115.997,-41.423,178.801,5.799,149.388
C04291=1166.837,-116.247,-41.415,178.800,5.799,149.389
C04292=1166.842,-116.497,-41.406,178.797,5.799,149.389
C04293=1166.848,-116.747,-41.396,178.795,5.799,149.390
C04294=1166.854,-116.996,-41.388,178.793,5.798,149.390
C04295=1166.859,-117.246,-41.379,178.791,5.799,149.391
C04296=1166.864,-117.496,-41.370,178.789,5.798,149.392
C04297=1166.869,-117.746,-41.361,178.787,5.798,149.392
C04298=1166.875,-117.995,-41.352,178.785,5.797,149.393
C04299=1166.880,-118.245,-41.343,178.783,5.797,149.393
C04300=1166.886,-118.494,-41.335,178.781,5.797,149.394
C04301=1166.891,-118.744,-41.326,178.779,5.797,149.394
C04302=1166.896,-118.994,-41.317,178.777,5.796,149.395
C04303=1166.901,-119.244,-41.308,178.775,5.796,149.395
C04304=1166.906,-119.494,-41.299,178.772,5.796,149.396
C04305=1166.913,-119.744,-41.291,178.771,5.796,149.397
C04306=1166.918,-119.994,-41.282,178.769,5.795,149.397
C04307=1166.923,-120.244,-41.273,178.767,5.795,149.398
C04308=1166.929,-120.493,-41.264,178.764,5.795,149.398
C04309=1166.934,-120.743,-41.255,178.763,5.795,149.399
C04310=1166.939,-120.992,-41.246,178.760,5.794,149.399
C04311=1166.945,-121.242,-41.238,178.758,5.795,149.400
C04312=1166.950,-121.492,-41.229,178.756,5.794,149.400
C04313=1166.955,-121.742,-41.220,178.755,5.794,149.401
C04314=1166.960,-121.993,-41.212,178.752,5.793,149.401
C04315=1166.966,-122.242,-41.203,178.750,5.794,149.402
C04316=1166.971,-122.492,-41.194,178.748,5.793,149.403
C04317=1166.977,-122.741,-41.185,178.746,5.793,149.403
C04318=1166.982,-122.991,-41.176,178.744,5.792,149.404
C04319=1166.987,-123.240,-41.168,178.742,5.792,149.404
C04320=1166.993,-123.491,-41.160,178.740,5.792,149.405
C04321=1166.998,-123.741,-41.151,178.738,5.792,149.406
C04322=1167.003,-123.991,-41.142,178.736,5.791,149.406
C04323=1167.009,-124.240,-41.133,178.734,5.791,149.406
C04324=1167.014,-124.490,-41.124,178.732,5.791,149.407
C04325=1167.020,-124.740,-41.116,178.730,5.791,149.408
C04326=1167.025,-124.990,-41.107,178.728,5.790,149.408
C04327=1167.031,-125.239,-41.099,178.726,5.790,149.409
C04328=1167.036,-125.489,-41.090,178.724,5.790,149.409
C04329=1167.041,-125.739,-41.082,178.722,5.790,149.410
C04330=1167.046,-125.989,-41.073,178.720,5.789,149.410
C04331=1167.051,-126.238,-41.065,178.718,5.789,149.411
C04332=1167.057,-126.488,-41.056,178.715,5.789,149.412
C04333=1167.062,-126.738,-41.048,178.714,5.789,149.412
C04334=1167.068,-126.987,-41.039,178.712,5.788,149.413
C04335=1167.073,-127.237,-41.030,178.710,5.788,149.413
C04336=1167.078,-127.487,-41.021,178.707,5.788,149.414
C04337=1167.084,-127.738,-41.013,178.706,5.788,149.414
C04338=1166.663,-127.749,-41.054,178.702,5.791,149.416
C04339=1166.657,-127.498,-41.063,178.704,5.791,149.415
C04340=1166.652,-127.249,-41.072,178.706,5.791,149.415
C04341=1166.646,-126.999,-41.080,178.708,5.791,149.414
C04342=1166.641,-126.749,-41.088,178.710,5.792,149.414
C04343=1166.636,-126.499,-41.097,178.712,5.792,149.413
C04344=1166.631,-126.249,-41.106,178.714,5.793,149.413
C04345=1166.625,-126.000,-41.115,178.716,5.793,149.412
C04346=1166.619,-125.750,-41.123,178.718,5.793,149.412
C04347=1166.614,-125.500,-41.132,178.720,5.793,149.411
C04348=1166.609,-125.250,-41.141,178.722,5.794,149.410
C04349=1166.603,-125.001,-41.149,178.724,5.794,149.410
C04350=1166.598,-124.750,-41.157,178.726,5.794,149.410
C04351=1166.593,-124.500,-41.166,178.728,5.794,149.409
C04352=1166.587,-124.251,-41.175,178.730,5.795,149.408
C04353=1166.582,-124.001,-41.184,178.732,5.795,149.408
C04354=1166.577,-123.752,-41.192,178.735,5.795,149.407
C04355=1166.572,-123.501,-41.200,178.736,5.795,149.407
C04356=1166.566,-123.252,-41.209,178.738,5.796,149.406
C04357=1166.561,-123.002,-41.218,178.740,5.796,149.406
C04358=1166.556,-122.753,-41.226,178.743,5.796,149.405
C04359=1166.551,-122.503,-41.235,178.744,5.796,149.404
C04360=1166.545,-122.253,-41.244,178.746,5.797,149.404
C04361=1166.539,-122.003,-41.252,178.748,5.797,149.403
C04362=1166.534,-121.753,-41.261,178.751,5.797,149.403
C04363=1166.529,-121.503,-41.270,178.752,5.797,149.402
C04364=1166.523,-121.253,-41.279,178.754,5.798,149.402
C04365=1166.517,-121.004,-41.288,178.757,5.797,149.401
C04366=1166.512,-120.754,-41.297,178.759,5.798,149.401
C04367=1166.507,-120.504,-41.306,178.760,5.798,149.400
C04368=1166.502,-120.255,-41.315,178.763,5.799,149.399
C04369=1166.496,-120.004,-41.323,178.765,5.799,149.399
C04370=1166.491,-119.755,-41.331,178.767,5.799,149.398
C04371=1166.485,-119.505,-41.340,178.768,5.799,149.398
C04372=1166.480,-119.255,-41.349,178.771,5.800,149.397
C04373=1166.475,-119.005,-41.358,178.773,5.800,149.397
C04374=1166.470,-118.755,-41.367,178.775,5.800,149.396
C04375=1166.465,-118.506,-41.376,178.778,5.801,149.396
C04376=1166.459,-118.257,-41.384,178.779,5.801,149.395
C04377=1166.454,-118.007,-41.393,178.781,5.801,149.395
C04378=1166.449,-117.757,-41.402,178.783,5.801,149.394
C04379=1166.444,-117.507,-41.411,178.786,5.802,149.393
C04380=1166.438,-117.257,-41.420,178.787,5.802,149.393
C04381=1166.432,-117.008,-41.429,178.789,5.803,149.392
C04382=1166.427,-116.758,-41.438,178.792,5.802,149.392
C04383=1166.422,-116.508,-41.447,178.794,5.803,149.391
C04384=1166.416,-116.258,-41.456,178.795,5.803,149.391
C04385=1166.411,-116.008,-41.465,178.798,5.803,149.390
C04386=1166.406,-115.758,-41.473,178.800,5.803,149.389
C04387=1166.401,-115.509,-41.482,178.802,5.804,149.389
C04388=1166.395,-115.259,-41.491,178.804,5.804,149.388
C04389=1166.389,-115.009,-41.500,178.806,5.804,149.388
C04390=1166.384,-114.759,-41.509,178.808,5.804,149.387
C04391=1166.379,-114.510,-41.518,178.810,5.805,149.387
C04392=1166.374,-114.260,-41.527,178.812,5.805,149.386
C04393=1166.369,-114.010,-41.536,178.814,5.805,149.386
C04394=1166.363,-113.760,-41.545,178.816,5.805,149.385
C04395=1166.357,-113.510,-41.554,178.818,5.806,149.384
C04396=1166.352,-113.261,-41.563,178.821,5.806,149.384
C04397=1166.346,-113.011,-41.572,178.823,5.806,149.383
C04398=1166.341,-112.761,-41.581,178.825,5.807,149.383
C04399=1166.336,-112.511,-41.590,178.826,5.807,149.382
C04400=1166.331,-112.261,-41.599,178.829,5.807,149.382
C04401=1166.325,-112.011,-41.608,178.831,5.807,149.381
C04402=1166.320,-111.762,-41.618,178.833,5.808,149.381
C04403=1166.315,-111.512,-41.627,178.835,5.807,149.380
C04404=1166.309,-111.263,-41.635,178.837,5.808,149.379
C04405=1166.303,-111.013,-41.645,178.839,5.808,149.379
C04406=1166.298,-110.763,-41.653,178.841,5.809,149.378
C04407=1166.293,-110.513,-41.662,178.844,5.809,149.378
C04408=1166.288,-110.263,-41.671,178.845,5.809,149.377
C04409=1166.283,-110.013,-41.680,178.848,5.810,149.376
C04410=1166.277,-109.764,-41.690,178.850,5.810,149.376
C04411=1166.272,-109.514,-41.699,178.852,5.810,149.376
C04412=1166.267,-109.264,-41.708,178.854,5.810,149.375
C04413=1166.262,-109.014,-41.717,178.856,5.811,149.374
C04414=1166.256,-108.764,-41.727,178.858,5.811,149.374
C04415=1166.251,-108.515,-41.736,178.860,5.811,149.373
C04416=1166.246,-108.265,-41.745,178.862,5.811,149.373
C04417=1166.241,-108.015,-41.754,178.865,5.811,149.372
C04418=1166.235,-107.765,-41.763,178.867,5.812,149.371
C04419=1166.229,-107.516,-41.772,178.868,5.812,149.371
C04420=1166.224,-107.267,-41.782,178.871,5.813,149.370
C04421=1166.218,-107.016,-41.791,178.873,5.813,149.370
C04422=1166.213,-106.767,-41.800,178.875,5.813,149.369
C04423=1166.208,-106.517,-41.809,178.877,5.813,149.369
C04424=1166.203,-106.267,-41.818,178.879,5.814,149.368
C04425=1166.197,-106.017,-41.828,178.881,5.814,149.368
C04426=1166.192,-105.767,-41.837,178.883,5.814,149.367
C04427=1166.187,-105.518,-41.846,178.886,5.815,149.366
C04428=1166.181,-105.268,-41.856,178.888,5.814,149.366
C04429=1166.176,-105.018,-41.865,178.890,5.815,149.365
C04430=1166.171,-104.768,-41.874,178.891,5.815,149.365
C04431=1166.165,-104.518,-41.883,178.894,5.816,149.364
C04432=1166.160,-104.269,-41.893,178.896,5.815,149.363
C04433=1166.155,-104.019,-41.902,178.898,5.816,149.363
C04434=1166.149,-103.769,-41.911,178.901,5.817,149.362
C04435=1166.144,-103.520,-41.921,178.902,5.817,149.362
C04436=1166.139,-103.270,-41.930,178.905,5.817,149.361
C04437=1166.133,-103.020,-41.939,178.906,5.817,149.361
C04438=1166.128,-102.770,-41.949,178.909,5.818,149.360
C04439=1166.123,-102.499,-41.959,178.911,5.818,149.359
C04440=1166.117,-102.227,-41.969,178.913,5.818,149.359
C04441=1166.111,-101.954,-41.980,178.916,5.818,149.358
C04442=1166.105,-101.682,-41.990,178.918,5.819,149.357
C04443=1166.100,-101.433,-41.999,178.920,5.819,149.357
C04444=1166.094,-101.182,-42.009,178.922,5.820,149.357
C04445=1166.089,-100.933,-42.018,178.924,5.819,149.356
C04446=1166.084,-100.683,-42.027,178.926,5.820,149.355
C04447=1166.078,-100.433,-42.037,178.929,5.820,149.355
C04448=1166.074,-100.184,-42.046,178.931,5.820,149.354
C04449=1166.068,-99.934,-42.056,178.933,5.821,149.354
C04450=1166.063,-99.685,-42.066,178.935,5.821,149.353
C04451=1166.057,-99.434,-42.075,178.937,5.821,149.352
C04452=1166.052,-99.185,-42.085,178.940,5.822,149.352
C04453=1166.047,-98.935,-42.094,178.941,5.822,149.351
C04454=1166.041,-98.685,-42.103,178.944,5.823,149.351
C04455=1166.036,-98.436,-42.113,178.946,5.822,149.350
C04456=1166.030,-98.186,-42.122,178.948,5.823,149.350
C04457=1166.025,-97.937,-42.132,178.950,5.823,149.349
C04458=1166.019,-97.686,-42.141,178.952,5.823,149.348
C04459=1166.015,-97.436,-42.151,178.954,5.824,149.348
C04460=1166.009,-97.186,-42.161,178.956,5.824,149.347
C04461=1166.004,-96.937,-42.170,178.959,5.824,149.347
C04462=1165.998,-96.687,-42.180,178.961,5.825,149.346
C04463=1165.994,-96.438,-42.189,178.963,5.825,149.345
C04464=1165.988,-96.187,-42.199,178.965,5.826,149.345
C04465=1165.983,-95.938,-42.209,178.967,5.825,149.344
C04466=1165.977,-95.688,-42.218,178.969,5.826,149.344
C04467=1165.972,-95.439,-42.228,178.972,5.826,149.343
C04468=1165.966,-95.189,-42.237,178.974,5.826,149.343
C04469=1165.962,-94.939,-42.247,178.976,5.827,149.342
C04470=1165.956,-94.689,-42.257,178.978,5.827,149.341
C04471=1165.951,-94.439,-42.266,178.980,5.827,149.341
C04472=1165.946,-94.190,-42.276,178.983,5.828,149.340
C04473=1165.940,-93.940,-42.285,178.984,5.828,149.340
C04474=1165.935,-93.690,-42.296,178.986,5.829,149.339
C04475=1165.929,-93.440,-42.305,178.989,5.828,149.339
C04476=1165.924,-93.191,-42.315,178.991,5.829,149.338
C04477=1165.919,-92.941,-42.325,178.993,5.829,149.337
C04478=1165.914,-92.691,-42.334,178.995,5.829,149.337
C04479=1165.908,-92.441,-42.344,178.998,5.830,149.336
C04480=1165.903,-92.192,-42.353,178.999,5.830,149.336
C04481=1165.898,-91.942,-42.363,179.001,5.830,149.335
C04482=1165.892,-91.692,-42.374,179.004,5.831,149.334
C04483=1165.887,-91.442,-42.383,179.006,5.831,149.334
C04484=1165.882,-91.192,-42.393,179.008,5.831,149.333
C04485=1165.877,-90.943,-42.403,179.011,5.832,149.333
C04486=1165.871,-90.693,-42.412,179.013,5.832,149.332
C04487=1165.865,-90.443,-42.422,179.015,5.832,149.332
C04488=1165.861,-90.194,-42.432,179.016,5.832,149.331
C04489=1165.855,-89.943,-42.442,179.019,5.833,149.330
C04490=1165.850,-89.694,-42.451,179.021,5.833,149.330
C04491=1165.845,-89.445,-42.462,179.023,5.833,149.329
C04492=1165.839,-89.194,-42.471,179.026,5.834,149.329
C04493=1165.834,-88.945,-42.481,179.028,5.834,149.328
C04494=1165.829,-88.695,-42.491,179.030,5.834,149.328
C04495=1165.823,-88.445,-42.502,179.032,5.835,149.327
C04496=1165.818,-88.196,-42.510,179.034,5.835,149.326
C04497=1165.813,-87.946,-42.521,179.036,5.835,149.326
C04498=1165.808,-87.696,-42.531,179.039,5.836,149.325
C04499=1165.803,-87.446,-42.541,179.041,5.836,149.325
C04500=1165.797,-87.196,-42.550,179.043,5.836,149.324
C04501=1165.791,-86.947,-42.561,179.045,5.837,149.323
C04502=1165.786,-86.698,-42.570,179.048,5.836,149.323
C04503=1165.781,-86.447,-42.581,179.050,5.837,149.322
C04504=1165.776,-86.197,-42.590,179.052,5.838,149.322
C04505=1165.771,-85.948,-42.600,179.054,5.838,149.321
C04506=1165.765,-85.698,-42.610,179.056,5.838,149.321
C04507=1165.760,-85.448,-42.621,179.059,5.839,149.320
C04508=1165.755,-85.199,-42.630,179.060,5.839,149.319
C04509=1165.750,-84.949,-42.640,179.063,5.839,149.319
C04510=1165.744,-84.699,-42.650,179.065,5.839,149.318
C04511=1165.739,-84.449,-42.661,179.067,5.840,149.318
C04512=1165.734,-84.200,-42.670,179.070,5.840,149.317
C04513=1165.728,-83.950,-42.680,179.071,5.840,149.317
C04514=1165.723,-83.700,-42.691,179.074,5.841,149.316
C04515=1165.718,-83.451,-42.701,179.076,5.841,149.315
C04516=1165.712,-83.201,-42.710,179.078,5.841,149.315
C04517=1165.707,-82.951,-42.720,179.080,5.842,149.314
C04518=1165.702,-82.701,-42.731,179.083,5.842,149.313
C04519=1165.697,-82.452,-42.740,179.085,5.842,149.313
C04520=1165.691,-82.202,-42.751,179.087,5.843,149.312
C04521=1165.686,-81.952,-42.761,179.089,5.843,149.312
C04522=1165.681,-81.702,-42.771,179.092,5.843,149.311
C04523=1165.675,-81.453,-42.782,179.094,5.844,149.311
C04524=1165.670,-81.203,-42.791,179.096,5.845,149.310
C04525=1165.665,-80.953,-42.802,179.098,5.844,149.309
C04526=1165.660,-80.704,-42.812,179.100,5.845,149.309
C04527=1165.654,-80.454,-42.822,179.103,5.845,149.308
C04528=1165.649,-80.203,-42.832,179.104,5.845,149.308
C04529=1165.644,-79.954,-42.842,179.107,5.846,149.307
C04530=1165.638,-79.704,-42.852,179.109,5.846,149.307
C04531=1165.633,-79.454,-42.863,179.111,5.846,149.306
C04532=1165.628,-79.205,-42.873,179.114,5.847,149.305
C04533=1165.622,-78.955,-42.883,179.116,5.847,149.305
C04534=1165.617,-78.705,-42.894,179.118,5.847,149.304
C04535=1165.612,-78.456,-42.903,179.121,5.848,149.303
C04536=1165.607,-78.206,-42.913,179.123,5.848,149.303
C04537=1165.602,-77.956,-42.924,179.125,5.848,149.302
C04538=1165.596,-77.706,-42.934,179.127,5.849,149.302
C04539=1165.591,-77.457,-42.944,179.130,5.849,149.301
C04540=1165.586,-77.206,-42.955,179.131,5.849,149.301
C04541=1165.580,-76.957,-42.965,179.133,5.850,149.300
C04542=1165.575,-76.708,-42.976,179.136,5.850,149.299
C04543=1165.569,-76.437,-42.987,179.139,5.851,149.299
C04544=1165.564,-76.165,-42.999,179.140,5.851,149.298
C04545=1165.558,-75.895,-43.009,179.143,5.851,149.297
C04546=1165.552,-75.623,-43.021,179.146,5.852,149.297
C04547=1165.546,-75.373,-43.031,179.148,5.852,149.296
C04548=1165.541,-75.123,-43.041,179.150,5.852,149.296
C04549=1165.536,-74.874,-43.052,179.152,5.853,149.295
C04550=1165.531,-74.624,-43.062,179.155,5.853,149.294
C04551=1165.526,-74.374,-43.072,179.157,5.854,149.294
C04552=1165.521,-74.125,-43.083,179.159,5.853,149.293
C04553=1165.516,-73.875,-43.093,179.161,5.854,149.293
C04554=1165.510,-73.625,-43.104,179.164,5.855,149.292
C04555=1165.505,-73.375,-43.114,179.166,5.855,149.292
C04556=1165.499,-73.126,-43.124,179.168,5.855,149.291
C04557=1165.494,-72.876,-43.134,179.170,5.856,149.290
C04558=1165.489,-72.626,-43.145,179.173,5.855,149.290
C04559=1165.483,-72.377,-43.156,179.175,5.856,149.289
C04560=1165.478,-72.127,-43.167,179.177,5.857,149.289
C04561=1165.473,-71.877,-43.177,179.179,5.857,149.288
C04562=1165.468,-71.627,-43.187,179.181,5.857,149.288
C04563=1165.462,-71.377,-43.198,179.184,5.858,149.287
C04564=1165.457,-71.128,-43.208,179.186,5.859,149.286
C04565=1165.452,-70.878,-43.219,179.188,5.858,149.286
C04566=1165.446,-70.629,-43.229,179.190,5.859,149.285
C04567=1165.441,-70.378,-43.240,179.193,5.859,149.284
C04568=1165.436,-70.129,-43.251,179.195,5.859,149.284
C04569=1165.431,-69.879,-43.261,179.197,5.860,149.283
C04570=1165.425,-69.630,-43.272,179.199,5.861,149.283
C04571=1165.420,-69.379,-43.282,179.202,5.861,149.282
C04572=1165.415,-69.131,-43.293,179.204,5.861,149.282
C04573=1165.410,-68.880,-43.304,179.206,5.861,149.281
C04574=1165.405,-68.631,-43.314,179.209,5.862,149.280
C04575=1165.399,-68.381,-43.324,179.211,5.862,149.280
C04576=1165.394,-68.132,-43.335,179.213,5.863,149.279
C04577=1165.388,-67.882,-43.346,179.215,5.863,149.278
C04578=1165.383,-67.631,-43.357,179.218,5.864,149.278
C04579=1165.378,-67.383,-43.368,179.220,5.863,149.277
C04580=1165.373,-67.132,-43.378,179.222,5.864,149.277
C04581=1165.367,-66.883,-43.388,179.225,5.864,149.276
C04582=1165.362,-66.633,-43.400,179.227,5.865,149.276
C04583=1165.357,-66.384,-43.410,179.229,5.865,149.275
C04584=1165.352,-66.133,-43.420,179.231,5.866,149.274
C04585=1165.346,-65.884,-43.431,179.234,5.866,149.274
C04586=1165.341,-65.634,-43.442,179.235,5.866,149.273
C04587=1165.336,-65.385,-43.452,179.238,5.866,149.273
C04588=1165.330,-65.135,-43.464,179.240,5.867,149.272
C04589=1165.325,-64.884,-43.475,179.243,5.868,149.271
C04590=1165.320,-64.636,-43.486,179.244,5.868,149.271
C04591=1165.315,-64.385,-43.496,179.247,5.868,149.270
C04592=1165.310,-64.136,-43.506,179.250,5.868,149.269
C04593=1165.305,-63.886,-43.518,179.252,5.869,149.269
C04594=1165.299,-63.637,-43.528,179.254,5.869,149.268
C04595=1165.294,-63.387,-43.540,179.256,5.870,149.268
C04596=1165.288,-63.137,-43.550,179.259,5.870,149.267
C04597=1165.284,-62.887,-43.561,179.261,5.871,149.267
C04598=1165.278,-62.638,-43.571,179.263,5.870,149.266
C04599=1165.273,-62.388,-43.582,179.265,5.871,149.265
C04600=1165.268,-62.138,-43.593,179.268,5.872,149.265
C04601=1165.262,-61.888,-43.604,179.270,5.872,149.264
C04602=1165.257,-61.639,-43.615,179.272,5.872,149.264
C04603=1165.252,-61.389,-43.626,179.274,5.873,149.263
C04604=1165.247,-61.139,-43.637,179.277,5.873,149.262
C04605=1165.242,-60.889,-43.647,179.279,5.874,149.262
C04606=1165.236,-60.640,-43.659,179.281,5.874,149.261
C04607=1165.231,-60.390,-43.670,179.284,5.874,149.261
C04608=1165.226,-60.141,-43.681,179.286,5.875,149.260
C04609=1165.221,-59.890,-43.691,179.288,5.876,149.260
C04610=1165.216,-59.641,-43.702,179.290,5.875,149.259
C04611=1165.210,-59.392,-43.714,179.293,5.876,149.258
C04612=1165.205,-59.141,-43.724,179.295,5.876,149.258
C04613=1165.200,-58.892,-43.735,179.298,5.877,149.257
C04614=1165.195,-58.642,-43.746,179.300,5.877,149.256
C04615=1165.189,-58.392,-43.758,179.302,5.878,149.256
C04616=1165.184,-58.143,-43.768,179.304,5.878,149.255
C04617=1165.179,-57.893,-43.779,179.307,5.879,149.255
C04618=1165.174,-57.643,-43.791,179.309,5.878,149.254
C04619=1165.168,-57.394,-43.801,179.311,5.879,149.253
C04620=1165.163,-57.144,-43.813,179.314,5.880,149.253
C04621=1165.158,-56.894,-43.823,179.316,5.880,149.252
C04622=1165.152,-56.645,-43.835,179.318,5.881,149.252
C04623=1165.147,-56.395,-43.846,179.320,5.880,149.251
C04624=1165.142,-56.145,-43.856,179.323,5.881,149.251
C04625=1165.137,-55.896,-43.868,179.325,5.882,149.250
C04626=1165.132,-55.646,-43.879,179.328,5.882,149.249
C04627=1165.126,-55.396,-43.890,179.330,5.882,149.249
C04628=1165.121,-55.147,-43.901,179.332,5.883,149.248
C04629=1165.116,-54.897,-43.913,179.334,5.883,149.247
C04630=1165.110,-54.647,-43.923,179.337,5.884,149.247
C04631=1165.106,-54.398,-43.934,179.339,5.884,149.246
C04632=1165.100,-54.148,-43.946,179.341,5.884,149.246
C04633=1165.096,-53.898,-43.958,179.344,5.885,149.245
C04634=1165.090,-53.648,-43.968,179.346,5.885,149.244
C04635=1165.085,-53.398,-43.980,179.348,5.886,149.244
C04636=1165.080,-53.149,-43.991,179.351,5.887,149.243
C04637=1165.074,-52.899,-44.002,179.353,5.887,149.243
C04638=1165.069,-52.649,-44.013,179.355,5.887,149.242
C04639=1165.064,-52.400,-44.024,179.358,5.888,149.242
C04640=1165.058,-52.151,-44.036,179.360,5.888,149.241
C04641=1165.053,-51.901,-44.047,179.362,5.888,149.240
C04642=1165.048,-51.651,-44.058,179.364,5.889,149.240
C04643=1165.043,-51.401,-44.070,179.367,5.889,149.239
C04644=1165.038,-51.152,-44.081,179.369,5.890,149.238
C04645=1165.032,-50.902,-44.092,179.372,5.891,149.238
C04646=1165.027,-50.652,-44.103,179.374,5.891,149.237
C04647=1165.021,-50.382,-44.116,179.376,5.891,149.237
C04648=1165.016,-50.111,-44.128,179.378,5.891,149.236
C04649=1165.010,-49.840,-44.140,179.381,5.892,149.235
C04650=1165.004,-49.570,-44.153,179.384,5.892,149.235
C04651=1165.000,-49.321,-44.164,179.386,5.893,149.234
C04652=1164.994,-49.070,-44.175,179.389,5.893,149.234
C04653=1164.989,-48.821,-44.186,179.391,5.894,149.233
C04654=1164.983,-48.571,-44.198,179.393,5.895,149.232
C04655=1164.978,-48.322,-44.209,179.396,5.894,149.232
C04656=1164.973,-48.072,-44.221,179.398,5.895,149.231
C04657=1164.968,-47.822,-44.232,179.400,5.895,149.230
C04658=1164.962,-47.573,-44.244,179.403,5.896,149.230
C04659=1164.958,-47.323,-44.255,179.405,5.897,149.229
C04660=1164.952,-47.073,-44.267,179.407,5.897,149.229
C04661=1164.947,-46.823,-44.278,179.409,5.897,149.228
C04662=1164.942,-46.573,-44.290,179.412,5.897,149.227
C04663=1164.936,-46.324,-44.300,179.414,5.898,149.227
C04664=1164.931,-46.074,-44.312,179.417,5.899,149.226
C04665=1164.926,-45.825,-44.324,179.419,5.900,149.226
C04666=1164.921,-45.575,-44.336,179.421,5.899,149.225
C04667=1164.916,-45.325,-44.347,179.423,5.900,149.225
C04668=1164.910,-45.076,-44.358,179.426,5.900,149.224
C04669=1164.905,-44.826,-44.370,179.428,5.901,149.223
C04670=1164.900,-44.576,-44.382,179.431,5.902,149.223
C04671=1164.895,-44.327,-44.393,179.433,5.902,149.222
C04672=1164.890,-44.077,-44.405,179.435,5.902,149.222
C04673=1164.884,-43.827,-44.416,179.438,5.902,149.221
C04674=1164.879,-43.578,-44.428,179.440,5.903,149.220
C04675=1164.874,-43.328,-44.439,179.443,5.904,149.220
C04676=1164.869,-43.078,-44.451,179.445,5.904,149.219
C04677=1164.864,-42.828,-44.463,179.448,5.905,149.218
C04678=1164.858,-42.578,-44.474,179.449,5.905,149.218
C04679=1164.854,-42.329,-44.486,179.452,5.905,149.217
C04680=1164.847,-42.080,-44.497,179.454,5.906,149.217
C04681=1164.843,-41.830,-44.509,179.457,5.907,149.216
C04682=1164.838,-41.581,-44.521,179.459,5.907,149.215
C04683=1164.832,-41.331,-44.533,179.462,5.908,149.215
C04684=1164.828,-41.081,-44.544,179.464,5.908,149.214
C04685=1164.822,-40.831,-44.556,179.466,5.908,149.214
C04686=1164.817,-40.581,-44.568,179.468,5.909,149.213
C04687=1164.812,-40.332,-44.579,179.471,5.909,149.213
C04688=1164.806,-40.082,-44.591,179.473,5.910,149.212
C04689=1164.801,-39.833,-44.602,179.475,5.911,149.211
C04690=1164.796,-39.583,-44.614,179.478,5.911,149.211
C04691=1164.791,-39.333,-44.627,179.481,5.911,149.210
C04692=1164.786,-39.084,-44.638,179.482,5.911,149.210
C04693=1164.781,-38.834,-44.650,179.485,5.912,149.209
C04694=1164.775,-38.584,-44.662,179.487,5.913,149.208
C04695=1164.770,-38.334,-44.674,179.490,5.913,149.208
C04696=1164.765,-38.084,-44.685,179.492,5.914,149.207
C04697=1164.759,-37.836,-44.697,179.495,5.914,149.207
C04698=1164.754,-37.586,-44.709,179.497,5.915,149.206
C04699=1164.749,-37.336,-44.720,179.499,5.915,149.205
C04700=1164.744,-37.086,-44.732,179.502,5.915,149.205
C04701=1164.739,-36.837,-44.745,179.504,5.916,149.204
C04702=1164.733,-36.587,-44.757,179.507,5.916,149.203
C04703=1164.729,-36.337,-44.768,179.509,5.917,149.203
C04704=1164.723,-36.087,-44.780,179.511,5.918,149.202
C04705=1164.718,-35.838,-44.792,179.514,5.918,149.202
C04706=1164.713,-35.588,-44.804,179.516,5.919,149.201
C04707=1164.708,-35.339,-44.816,179.518,5.918,149.200
C04708=1164.702,-35.089,-44.828,179.520,5.919,149.200
C04709=1164.697,-34.839,-44.840,179.523,5.920,149.199
C04710=1164.692,-34.589,-44.852,179.525,5.921,149.199
C04711=1164.687,-34.340,-44.863,179.528,5.921,149.198
C04712=1164.682,-34.090,-44.876,179.530,5.922,149.198
C04713=1164.677,-33.840,-44.888,179.533,5.922,149.197
C04714=1164.671,-33.591,-44.900,179.535,5.923,149.196
C04715=1164.666,-33.341,-44.912,179.538,5.923,149.196
C04716=1164.661,-33.092,-44.924,179.540,5.923,149.195
C04717=1164.656,-32.842,-44.935,179.542,5.924,149.195
C04718=1164.651,-32.592,-44.948,179.545,5.924,149.194
C04719=1164.645,-32.342,-44.960,179.547,5.925,149.193
C04720=1164.640,-32.092,-44.972,179.549,5.926,149.193
C04721=1164.635,-31.843,-44.984,179.552,5.926,149.192
C04722=1164.630,-31.594,-44.996,179.554,5.927,149.192
C04723=1164.625,-31.344,-45.008,179.557,5.927,149.191
C04724=1164.620,-31.094,-45.020,179.559,5.928,149.190
C04725=1164.614,-30.844,-45.032,179.561,5.928,149.190
C04726=1164.609,-30.595,-45.045,179.563,5.928,149.189
C04727=1164.604,-30.345,-45.057,179.566,5.929,149.188
C04728=1164.598,-30.096,-45.069,179.568,5.930,149.188
C04729=1164.594,-29.846,-45.080,179.571,5.930,149.187
C04730=1164.588,-29.596,-45.092,179.574,5.931,149.187
C04731=1164.583,-29.347,-45.105,179.576,5.931,149.186
C04732=1164.578,-29.097,-45.117,179.578,5.932,149.185
C04733=1164.573,-28.848,-45.129,179.581,5.933,149.185
C04734=1164.567,-28.598,-45.141,179.583,5.933,149.184
C04735=1164.562,-28.348,-45.154,179.585,5.934,149.184
C04736=1164.557,-28.098,-45.166,179.588,5.934,149.183
C04737=1164.552,-27.849,-45.178,179.590,5.934,149.182
C04738=1164.546,-27.599,-45.190,179.592,5.935,149.182
C04739=1164.541,-27.350,-45.203,179.595,5.935,149.181
C04740=1164.536,-27.100,-45.214,179.597,5.936,149.181
C04741=1164.532,-26.850,-45.227,179.600,5.936,149.180
C04742=1164.527,-26.601,-45.240,179.602,5.937,149.180
C04743=1164.521,-26.351,-45.252,179.605,5.938,149.179
C04744=1164.516,-26.102,-45.264,179.607,5.938,149.178
C04745=1164.511,-25.852,-45.276,179.609,5.939,149.178
C04746=1164.506,-25.602,-45.289,179.612,5.939,149.177
C04747=1164.500,-25.352,-45.301,179.614,5.940,149.177
C04748=1164.495,-25.103,-45.313,179.617,5.941,149.176
C04749=1164.490,-24.854,-45.326,179.619,5.941,149.175
C04750=1164.485,-24.603,-45.338,179.621,5.941,149.175
C04751=1164.479,-24.334,-45.351,179.625,5.942,149.174
C04752=1164.473,-24.064,-45.365,179.627,5.943,149.173
C04753=1164.468,-23.794,-45.378,179.629,5.943,149.173
C04754=1164.463,-23.524,-45.391,179.632,5.944,149.172
C04755=1164.457,-23.275,-45.404,179.635,5.944,149.171
C04756=1164.452,-23.026,-45.416,179.637,5.945,149.171
C04757=1164.446,-22.775,-45.429,179.640,5.946,149.170
C04758=1164.442,-22.525,-45.442,179.642,5.946,149.170
C04759=1164.436,-22.276,-45.454,179.644,5.947,149.169
C04760=1164.431,-22.026,-45.466,179.647,5.948,149.169
C04761=1164.426,-21.777,-45.479,179.649,5.947,149.168
C04762=1164.421,-21.527,-45.492,179.651,5.948,149.167
C04763=1164.415,-21.277,-45.503,179.653,5.948,149.167
C04764=1164.411,-21.027,-45.516,179.656,5.949,149.166
C04765=1164.406,-20.778,-45.529,179.658,5.950,149.166
C04766=1164.401,-20.529,-45.542,179.661,5.950,149.165
C04767=1164.395,-20.279,-45.554,179.664,5.951,149.164
C04768=1164.390,-20.029,-45.566,179.666,5.951,149.164
C04769=1164.384,-19.780,-45.579,179.668,5.952,149.163
C04770=1164.380,-19.530,-45.592,179.671,5.953,149.163
C04771=1164.374,-19.280,-45.604,179.673,5.953,149.162
C04772=1164.369,-19.031,-45.617,179.675,5.954,149.161
C04773=1164.364,-18.781,-45.629,179.678,5.954,149.161
C04774=1164.359,-18.532,-45.642,179.681,5.955,149.160
C04775=1164.354,-18.282,-45.655,179.683,5.956,149.160
C04776=1164.349,-18.032,-45.667,179.686,5.956,149.159
C04777=1164.343,-17.782,-45.680,179.688,5.957,149.158
C04778=1164.338,-17.533,-45.693,179.690,5.957,149.158
C04779=1164.333,-17.283,-45.706,179.693,5.958,149.157
C04780=1164.328,-17.034,-45.718,179.695,5.959,149.157
C04781=1164.323,-16.784,-45.731,179.698,5.959,149.156
C04782=1164.318,-16.535,-45.743,179.700,5.960,149.155
C04783=1164.312,-16.285,-45.756,179.703,5.960,149.155
C04784=1164.307,-16.035,-45.769,179.705,5.961,149.154
C04785=1164.302,-15.786,-45.781,179.708,5.962,149.154
C04786=1164.297,-15.536,-45.794,179.710,5.962,149.153
C04787=1164.293,-15.286,-45.807,179.712,5.963,149.152
C04788=1164.287,-15.037,-45.820,179.715,5.963,149.152
C04789=1164.282,-14.787,-45.833,179.717,5.964,149.151
C04790=1164.276,-14.538,-45.845,179.720,5.964,149.151
C04791=1164.272,-14.288,-45.858,179.722,5.965,149.150
C04792=1164.266,-14.038,-45.872,179.725,5.966,149.149
C04793=1164.261,-13.789,-45.884,179.727,5.967,149.149
C04794=1164.256,-13.540,-45.897,179.730,5.967,149.148
C04795=1164.251,-13.290,-45.910,179.732,5.967,149.148
C04796=1164.245,-13.040,-45.923,179.734,5.968,149.147
C04797=1164.240,-12.791,-45.936,179.737,5.969,149.146
C04798=1164.236,-12.541,-45.948,179.739,5.970,149.146
C04799=1164.231,-12.291,-45.961,179.742,5.970,149.145
C04800=1164.225,-12.042,-45.974,179.744,5.971,149.145
C04801=1164.220,-11.792,-45.987,179.747,5.971,149.144
C04802=1164.215,-11.542,-46.000,179.749,5.972,149.143
C04803=1164.209,-11.293,-46.013,179.752,5.972,149.143
C04804=1164.205,-11.043,-46.026,179.754,5.973,149.142
C04805=1164.200,-10.793,-46.039,179.756,5.974,149.142
C04806=1164.194,-10.544,-46.052,179.759,5.974,149.141
C04807=1164.189,-10.294,-46.065,179.761,5.975,149.141
C04808=1164.184,-10.044,-46.077,179.764,5.975,149.140
C04809=1164.179,-9.795,-46.090,179.767,5.976,149.139
C04810=1164.174,-9.545,-46.104,179.769,5.977,149.139
C04811=1164.169,-9.295,-46.116,179.771,5.977,149.138
C04812=1164.163,-9.046,-46.129,179.774,5.978,149.138
C04813=1164.159,-8.796,-46.143,179.776,5.978,149.137
C04814=1164.153,-8.547,-46.156,179.779,5.979,149.136
C04815=1164.148,-8.297,-46.169,179.781,5.980,149.136
C04816=1164.143,-8.047,-46.182,179.784,5.980,149.135
C04817=1164.138,-7.798,-46.194,179.786,5.981,149.135
C04818=1164.133,-7.548,-46.208,179.789,5.981,149.134
C04819=1164.128,-7.298,-46.221,179.791,5.982,149.133
C04820=1164.122,-7.049,-46.234,179.793,5.983,149.133
C04821=1164.117,-6.799,-46.247,179.796,5.983,149.132
C04822=1164.112,-6.550,-46.260,179.798,5.984,149.132
C04823=1164.107,-6.300,-46.274,179.801,5.984,149.131
C04824=1164.102,-6.051,-46.286,179.803,5.985,149.130
C04825=1164.096,-5.802,-46.300,179.806,5.986,149.130
C04826=1164.092,-5.551,-46.313,179.808,5.987,149.129
C04827=1164.086,-5.302,-46.326,179.811,5.987,149.129
C04828=1164.081,-5.052,-46.339,179.813,5.987,149.128
C04829=1164.077,-4.803,-46.353,179.815,5.988,149.127
C04830=1164.071,-4.554,-46.366,179.818,5.989,149.127
C04831=1164.066,-4.303,-46.379,179.820,5.990,149.126
C04832=1164.060,-4.054,-46.392,179.823,5.990,149.126
C04833=1164.056,-3.804,-46.406,179.826,5.992,149.125
C04834=1164.050,-3.555,-46.419,179.828,5.992,149.124
C04835=1164.046,-3.305,-46.432,179.831,5.992,149.124
C04836=1164.040,-3.056,-46.446,179.833,5.993,149.123
C04837=1164.036,-2.806,-46.459,179.836,5.994,149.123
C04838=1164.030,-2.556,-46.472,179.838,5.995,149.122
C04839=1164.025,-2.307,-46.485,179.841,5.995,149.121
C04840=1164.020,-2.057,-46.499,179.843,5.996,149.121
C04841=1164.015,-1.808,-46.511,179.845,5.996,149.120
C04842=1164.010,-1.558,-46.526,179.848,5.997,149.120
C04843=1164.005,-1.309,-46.538,179.850,5.998,149.119
C04844=1163.999,-1.058,-46.552,179.853,5.998,149.118
C04845=1163.994,-0.809,-46.566,179.855,5.999,149.118
C04846=1163.989,-0.559,-46.579,179.858,5.999,149.117
C04847=1163.984,-0.310,-46.593,179.860,6.000,149.117
C04848=1163.979,-0.060,-46.605,179.863,6.001,149.116
C04849=1163.973,0.189,-46.619,179.866,6.002,149.115
C04850=1163.969,0.439,-46.632,179.868,6.003,149.115
C04851=1163.963,0.688,-46.646,179.871,6.003,149.114
C04852=1163.958,0.938,-46.660,179.873,6.004,149.114
C04853=1163.953,1.187,-46.672,179.875,6.004,149.113
C04854=1163.948,1.437,-46.687,179.878,6.005,149.113
C04855=1163.942,1.707,-46.701,179.880,6.006,149.112
C04856=1163.937,1.975,-46.715,179.883,6.006,149.111
C04857=1163.932,2.245,-46.730,179.886,6.007,149.111
C04858=1163.926,2.514,-46.745,179.889,6.008,149.110
C04859=1163.920,2.764,-46.758,179.891,6.009,149.109
C04860=1163.916,3.013,-46.772,179.894,6.009,149.109
C04861=1163.910,3.263,-46.785,179.896,6.010,149.108
C04862=1163.906,3.512,-46.799,179.899,6.010,149.108
C04863=1163.900,3.762,-46.812,179.901,6.011,149.107
C04864=1163.895,4.012,-46.826,179.903,6.012,149.106
C04865=1163.891,4.262,-46.839,179.906,6.013,149.106
C04866=1163.885,4.511,-46.853,179.909,6.014,149.105
C04867=1163.880,4.761,-46.867,179.911,6.014,149.105
C04868=1163.875,5.010,-46.880,179.914,6.015,149.104
C04869=1163.870,5.259,-46.894,179.916,6.016,149.103
C04870=1163.865,5.510,-46.908,179.918,6.016,149.103
C04871=1163.859,5.759,-46.922,179.921,6.017,149.102
C04872=1163.855,6.009,-46.935,179.923,6.018,149.102
C04873=1163.849,6.258,-46.949,179.926,6.018,149.101
C04874=1163.844,6.508,-46.963,179.929,6.019,149.100
C04875=1163.840,6.758,-46.976,179.931,6.020,149.100
C04876=1163.834,7.007,-46.990,179.934,6.021,149.099
C04877=1163.829,7.256,-47.004,179.936,6.021,149.099
C04878=1163.823,7.506,-47.017,179.939,6.022,149.098
C04879=1163.819,7.755,-47.031,179.941,6.023,149.098
C04880=1163.814,8.005,-47.045,179.944,6.023,149.097
C04881=1163.808,8.255,-47.058,179.946,6.024,149.096
C04882=1163.803,8.504,-47.073,179.948,6.025,149.096
C04883=1163.799,8.754,-47.086,179.952,6.026,149.095
C04884=1163.794,9.003,-47.100,179.954,6.027,149.095
C04885=1163.788,9.253,-47.114,179.956,6.027,149.094
C04886=1163.783,9.502,-47.128,179.959,6.028,149.094
C04887=1163.778,9.752,-47.142,179.961,6.028,149.093
C04888=1163.774,10.001,-47.156,179.964,6.029,149.092
C04889=1163.768,10.251,-47.169,179.966,6.030,149.092
C04890=1163.763,10.501,-47.183,179.969,6.030,149.091
C04891=1163.758,10.750,-47.197,179.972,6.032,149.091
C04892=1163.752,10.999,-47.211,179.974,6.032,149.090
C04893=1163.747,11.250,-47.225,179.976,6.033,149.089
C04894=1163.743,11.499,-47.239,179.979,6.034,149.089
C04895=1163.737,11.748,-47.253,179.981,6.034,149.088
C04896=1163.732,11.998,-47.267,179.984,6.035,149.088
C04897=1163.727,12.247,-47.281,179.986,6.035,149.087
C04898=1163.722,12.497,-47.295,179.989,6.037,149.087
C04899=1163.717,12.747,-47.309,179.992,6.037,149.086
C04900=1163.712,12.996,-47.323,179.994,6.038,149.085
C04901=1163.707,13.246,-47.337,179.997,6.039,149.085
C04902=1163.702,13.495,-47.350,179.999,6.040,149.084
C04903=1163.697,13.745,-47.365,-179.998,6.040,149.084
C04904=1163.692,13.994,-47.379,-179.996,6.041,149.083
C04905=1163.687,14.244,-47.393,-179.993,6.042,149.082
C04906=1163.681,14.493,-47.407,-179.990,6.043,149.082
C04907=1163.676,14.743,-47.421,-179.988,6.043,149.081
C04908=1163.671,14.993,-47.435,-179.986,6.044,149.081
C04909=1163.666,15.242,-47.449,-179.983,6.045,149.080
C04910=1163.661,15.492,-47.463,-179.981,6.045,149.079
C04911=1163.656,15.741,-47.477,-179.978,6.047,149.079
C04912=1163.651,15.991,-47.492,-179.975,6.047,149.078
C04913=1163.645,16.240,-47.506,-179.973,6.048,149.078
C04914=1163.640,16.490,-47.520,-179.971,6.049,149.077
C04915=1163.635,16.740,-47.534,-179.968,6.049,149.076
C04916=1163.630,16.989,-47.548,-179.966,6.050,149.076
C04917=1163.625,17.239,-47.563,-179.962,6.051,149.075
C04918=1163.620,17.488,-47.577,-179.960,6.052,149.075
C04919=1163.615,17.738,-47.591,-179.958,6.052,149.074
C04920=1163.610,17.987,-47.605,-179.956,6.053,149.074
C04921=1163.605,18.237,-47.620,-179.953,6.054,149.073
C04922=1163.600,18.487,-47.634,-179.951,6.055,149.073
C04923=1163.595,18.736,-47.648,-179.947,6.056,149.072
C04924=1163.590,18.986,-47.662,-179.945,6.056,149.071
C04925=1163.585,19.235,-47.676,-179.943,6.057,149.071
C04926=1163.580,19.484,-47.691,-179.940,6.058,149.070
C04927=1163.575,19.734,-47.706,-179.938,6.058,149.070
C04928=1163.569,19.983,-47.719,-179.935,6.060,149.069
C04929=1163.565,20.233,-47.734,-179.932,6.061,149.069
C04930=1163.560,20.483,-47.748,-179.930,6.061,149.068
C04931=1163.555,20.732,-47.762,-179.928,6.062,149.067
C04932=1163.550,20.982,-47.777,-179.925,6.062,149.067
C04933=1163.545,21.232,-47.791,-179.922,6.064,149.066
C04934=1163.539,21.480,-47.805,-179.920,6.064,149.066
C04935=1163.534,21.730,-47.820,-179.917,6.065,149.065
C04936=1163.530,21.979,-47.834,-179.915,6.066,149.064
C04937=1163.525,22.229,-47.848,-179.912,6.066,149.064
C04938=1163.519,22.479,-47.863,-179.909,6.068,149.063
C04939=1163.514,22.729,-47.877,-179.907,6.068,149.063
C04940=1163.509,22.978,-47.892,-179.905,6.069,149.062
C04941=1163.504,23.227,-47.906,-179.902,6.070,149.061
C04942=1163.499,23.477,-47.921,-179.900,6.071,149.061
C04943=1163.494,23.726,-47.935,-179.896,6.072,149.060
C04944=1163.489,23.976,-47.950,-179.894,6.072,149.060
C04945=1163.483,24.226,-47.965,-179.892,6.073,149.059
C04946=1163.479,24.475,-47.979,-179.889,6.074,149.059
C04947=1163.474,24.725,-47.993,-179.886,6.075,149.058
C04948=1163.469,24.974,-48.008,-179.884,6.076,149.057
C04949=1163.464,25.224,-48.023,-179.881,6.077,149.057
C04950=1163.458,25.473,-48.036,-179.879,6.077,149.056
C04951=1163.453,25.723,-48.051,-179.877,6.078,149.056
C04952=1163.448,25.972,-48.066,-179.873,6.079,149.055
C04953=1163.443,26.222,-48.081,-179.871,6.080,149.055
C04954=1163.438,26.471,-48.095,-179.869,6.080,149.054
C04955=1163.434,26.720,-48.110,-179.866,6.081,149.054
C04956=1163.428,26.970,-48.125,-179.863,6.083,149.053
C04957=1163.423,27.220,-48.139,-179.861,6.083,149.052
C04958=1163.418,27.469,-48.154,-179.858,6.084,149.052
C04959=1163.412,27.738,-48.170,-179.856,6.084,149.051
C04960=1163.407,28.007,-48.186,-179.852,6.086,149.050
C04961=1163.402,28.276,-48.202,-179.850,6.086,149.050
C04962=1163.396,28.545,-48.218,-179.847,6.088,149.049
C04963=1163.391,28.795,-48.232,-179.844,6.088,149.049
C04964=1163.386,29.044,-48.247,-179.842,6.089,149.048
C04965=1163.381,29.293,-48.261,-179.840,6.090,149.047
C04966=1163.375,29.543,-48.276,-179.837,6.091,149.047
C04967=1163.371,29.792,-48.291,-179.834,6.092,149.046
C04968=1163.366,30.042,-48.305,-179.832,6.093,149.046
C04969=1163.360,30.291,-48.321,-179.829,6.093,149.045
C04970=1163.355,30.541,-48.335,-179.827,6.095,149.045
C04971=1163.351,30.790,-48.350,-179.824,6.095,149.044
C04972=1163.345,31.040,-48.365,-179.822,6.096,149.044
C04973=1163.340,31.289,-48.380,-179.819,6.096,149.043
C04974=1163.335,31.539,-48.394,-179.816,6.098,149.042
C04975=1163.330,31.788,-48.410,-179.814,6.099,149.042
C04976=1163.325,32.038,-48.424,-179.812,6.099,149.041
C04977=1163.320,32.287,-48.439,-179.809,6.100,149.041
C04978=1163.315,32.538,-48.454,-179.806,6.102,149.040
C04979=1163.311,32.787,-48.469,-179.804,6.102,149.040
C04980=1163.306,33.036,-48.484,-179.801,6.103,149.039
C04981=1163.300,33.286,-48.499,-179.798,6.104,149.038
C04982=1163.295,33.536,-48.514,-179.796,6.105,149.038
C04983=1163.290,33.785,-48.529,-179.793,6.105,149.037
C04984=1163.285,34.034,-48.544,-179.791,6.106,149.037
C04985=1163.280,34.284,-48.558,-179.788,6.108,149.036
C04986=1163.275,34.533,-48.574,-179.785,6.108,149.036
C04987=1163.270,34.782,-48.589,-179.783,6.109,149.035
C04988=1163.265,35.032,-48.604,-179.781,6.109,149.034
C04989=1163.260,35.281,-48.619,-179.778,6.111,149.034
C04990=1163.255,35.531,-48.633,-179.775,6.112,149.033
C04991=1163.250,35.780,-48.649,-179.773,6.112,149.033
C04992=1163.245,36.030,-48.664,-179.770,6.114,149.032
C04993=1163.239,36.280,-48.679,-179.768,6.115,149.032
C04994=1163.235,36.529,-48.694,-179.765,6.115,149.031
C04995=1163.230,36.779,-48.710,-179.762,6.117,149.031
C04996=1163.225,37.028,-48.725,-179.760,6.117,149.030
C04997=1163.220,37.278,-48.739,-179.757,6.118,149.029
C04998=1163.215,37.527,-48.754,-179.755,6.119,149.029
C04999=1163.210,37.776,-48.770,-179.752,6.120,149.028
C05000=1163.205,38.026,-48.784,-179.749,6.121,149.028
C05001=1163.199,38.275,-48.800,-179.747,6.121,149.027
C05002=1163.195,38.525,-48.815,-179.744,6.123,149.027
C05003=1163.189,38.774,-48.830,-179.742,6.124,149.026
C05004=1163.185,39.024,-48.846,-179.739,6.124,149.025
C05005=1163.179,39.274,-48.861,-179.736,6.126,149.025
C05006=1163.175,39.523,-48.876,-179.734,6.126,149.024
C05007=1163.169,39.772,-48.891,-179.731,6.127,149.024
C05008=1163.164,40.022,-48.907,-179.729,6.128,149.023
C05009=1163.159,40.271,-48.922,-179.726,6.129,149.022
C05010=1163.154,40.522,-48.937,-179.724,6.130,149.022
C05011=1163.150,40.771,-48.952,-179.721,6.130,149.021
C05012=1163.144,41.020,-48.968,-179.718,6.132,149.021
C05013=1163.140,41.269,-48.983,-179.716,6.132,149.020
C05014=1163.134,41.518,-48.998,-179.713,6.133,149.020
C05015=1163.129,41.768,-49.014,-179.710,6.135,149.019
C05016=1163.125,42.018,-49.029,-179.708,6.135,149.019
C05017=1163.119,42.267,-49.045,-179.705,6.136,149.018
C05018=1163.114,42.517,-49.060,-179.703,6.138,149.018
C05019=1163.109,42.766,-49.075,-179.700,6.138,149.017
C05020=1163.104,43.016,-49.090,-179.698,6.139,149.016
C05021=1163.100,43.265,-49.106,-179.695,6.140,149.016
C05022=1163.094,43.515,-49.121,-179.692,6.141,149.015
C05023=1163.089,43.764,-49.137,-179.690,6.141,149.015
C05024=1163.084,44.013,-49.152,-179.687,6.143,149.014
C05025=1163.079,44.263,-49.167,-179.684,6.144,149.014
C05026=1163.074,44.513,-49.183,-179.682,6.144,149.013
C05027=1163.069,44.762,-49.198,-179.679,6.146,149.012
C05028=1163.064,45.011,-49.214,-179.677,6.147,149.012
C05029=1163.059,45.261,-49.229,-179.674,6.147,149.011
C05030=1163.055,45.510,-49.245,-179.671,6.149,149.011
C05031=1163.049,45.760,-49.260,-179.669,6.149,149.010
C05032=1163.044,46.009,-49.276,-179.667,6.150,149.010
C05033=1163.038,46.259,-49.292,-179.663,6.151,149.009
C05034=1163.034,46.508,-49.307,-179.661,6.152,149.009
C05035=1163.029,46.758,-49.323,-179.658,6.154,149.008
C05036=1163.024,47.007,-49.338,-179.656,6.154,149.008
C05037=1163.019,47.256,-49.353,-179.653,6.155,149.007
C05038=1163.014,47.506,-49.370,-179.650,6.157,149.006
C05039=1163.009,47.755,-49.385,-179.648,6.157,149.006
C05040=1163.004,48.005,-49.401,-179.646,6.158,149.005
C05041=1163.000,48.254,-49.416,-179.643,6.160,149.005
C05042=1162.994,48.504,-49.432,-179.640,6.160,149.004
C05043=1162.989,48.753,-49.448,-179.638,6.161,149.004
C05044=1162.984,49.003,-49.463,-179.635,6.162,149.003
C05045=1162.979,49.253,-49.479,-179.633,6.163,149.003
C05046=1162.974,49.501,-49.495,-179.630,6.164,149.002
C05047=1162.970,49.751,-49.511,-179.627,6.165,149.002
C05048=1162.964,50.001,-49.526,-179.625,6.166,149.001
C05049=1162.959,50.250,-49.542,-179.622,6.167,149.000
C05050=1162.954,50.500,-49.558,-179.619,6.168,149.000
C05051=1162.950,50.749,-49.574,-179.617,6.169,148.999
C05052=1162.944,50.998,-49.589,-179.614,6.170,148.999
C05053=1162.939,51.248,-49.605,-179.612,6.171,148.998
C05054=1162.934,51.498,-49.621,-179.609,6.172,148.998
C05055=1162.929,51.746,-49.637,-179.606,6.173,148.997
C05056=1162.924,51.997,-49.653,-179.604,6.174,148.996
C05057=1162.919,52.246,-49.669,-179.601,6.175,148.996
C05058=1162.914,52.495,-49.684,-179.598,6.176,148.995
C05059=1162.910,52.745,-49.700,-179.596,6.177,148.995
C05060=1162.904,52.994,-49.716,-179.593,6.178,148.994
C05061=1162.899,53.243,-49.731,-179.591,6.179,148.994
C05062=1162.894,53.493,-49.748,-179.588,6.180,148.993
C05063=1162.889,53.761,-49.765,-179.586,6.181,148.993
C05064=1162.883,54.030,-49.782,-179.582,6.182,148.992
C05065=1162.878,54.299,-49.799,-179.579,6.184,148.991
C05066=1162.873,54.567,-49.816,-179.577,6.184,148.991
C05067=1162.867,54.817,-49.832,-179.574,6.186,148.990
C05068=1162.863,55.066,-49.849,-179.572,6.187,148.990
C05069=1162.858,55.316,-49.864,-179.569,6.187,148.989
C05070=1162.853,55.564,-49.881,-179.566,6.189,148.989
C05071=1162.848,55.815,-49.897,-179.564,6.190,148.988
C05072=1162.842,56.064,-49.912,-179.561,6.191,148.988
C05073=1162.838,56.313,-49.929,-179.559,6.192,148.987
C05074=1162.832,56.563,-49.944,-179.556,6.192,148.986
C05075=1162.828,56.812,-49.961,-179.553,6.194,148.986
C05076=1162.823,57.062,-49.977,-179.551,6.194,148.985
C05077=1162.818,57.311,-49.993,-179.548,6.196,148.985
C05078=1162.813,57.561,-50.009,-179.545,6.197,148.984
C05079=1162.808,57.809,-50.025,-179.542,6.198,148.984
C05080=1162.803,58.060,-50.041,-179.540,6.199,148.983
C05081=1162.798,58.308,-50.057,-179.538,6.200,148.983
C05082=1162.793,58.558,-50.073,-179.534,6.201,148.982
C05083=1162.788,58.807,-50.090,-179.532,6.202,148.982
C05084=1162.783,59.057,-50.106,-179.530,6.203,148.981
C05085=1162.778,59.306,-50.122,-179.527,6.204,148.981
C05086=1162.773,59.556,-50.138,-179.524,6.206,148.980
C05087=1162.768,59.805,-50.154,-179.522,6.206,148.979
C05088=1162.763,60.055,-50.170,-179.519,6.207,148.979
C05089=1162.758,60.304,-50.187,-179.516,6.208,148.978
C05090=1162.754,60.554,-50.202,-179.514,6.209,148.978
C05091=1162.748,60.803,-50.219,-179.511,6.210,148.977
C05092=1162.743,61.053,-50.236,-179.509,6.211,148.977
C05093=1162.738,61.302,-50.252,-179.505,6.213,148.976
C05094=1162.733,61.551,-50.268,-179.503,6.214,148.976
C05095=1162.728,61.800,-50.285,-179.501,6.215,148.975
C05096=1162.723,62.050,-50.301,-179.498,6.216,148.975
C05097=1162.718,62.299,-50.317,-179.495,6.217,148.974
C05098=1162.714,62.549,-50.333,-179.493,6.218,148.973
C05099=1162.709,62.798,-50.349,-179.490,6.219,148.973
C05100=1162.703,63.048,-50.366,-179.487,6.220,148.972
C05101=1162.699,63.297,-50.383,-179.485,6.221,148.972
C05102=1162.693,63.547,-50.399,-179.482,6.223,148.972
C05103=1162.689,63.796,-50.415,-179.480,6.223,148.971
C05104=1162.684,64.045,-50.432,-179.477,6.225,148.970
C05105=1162.679,64.295,-50.448,-179.474,6.225,148.970
C05106=1162.673,64.544,-50.464,-179.472,6.227,148.969
C05107=1162.669,64.794,-50.481,-179.469,6.227,148.969
C05108=1162.664,65.043,-50.498,-179.466,6.229,148.968
C05109=1162.659,65.293,-50.513,-179.464,6.230,148.968
C05110=1162.654,65.542,-50.531,-179.461,6.231,148.967
C05111=1162.649,65.791,-50.547,-179.459,6.232,148.967
C05112=1162.644,66.041,-50.564,-179.455,6.234,148.966
C05113=1162.640,66.290,-50.580,-179.453,6.234,148.966
C05114=1162.634,66.539,-50.596,-179.450,6.236,148.965
C05115=1162.629,66.789,-50.613,-179.448,6.237,148.965
C05116=1162.624,67.038,-50.629,-179.445,6.238,148.964
C05117=1162.620,67.288,-50.646,-179.443,6.239,148.963
C05118=1162.615,67.537,-50.663,-179.440,6.240,148.963
C05119=1162.609,67.786,-50.680,-179.437,6.241,148.962
C05120=1162.605,68.036,-50.696,-179.434,6.243,148.962
C05121=1162.600,68.286,-50.712,-179.432,6.243,148.961
C05122=1162.594,68.535,-50.729,-179.429,6.245,148.961
C05123=1162.590,68.784,-50.746,-179.426,6.245,148.960
C05124=1162.585,69.034,-50.763,-179.424,6.247,148.960
C05125=1162.579,69.283,-50.779,-179.422,6.248,148.959
C05126=1162.575,69.532,-50.796,-179.418,6.249,148.959
C05127=1162.570,69.782,-50.813,-179.416,6.250,148.958
C05128=1162.565,70.031,-50.830,-179.413,6.251,148.958
C05129=1162.560,70.280,-50.846,-179.411,6.252,148.957
C05130=1162.556,70.530,-50.863,-179.408,6.254,148.957
C05131=1162.550,70.779,-50.880,-179.405,6.254,148.956
C05132=1162.545,71.028,-50.897,-179.403,6.256,148.956
C05133=1162.541,71.278,-50.913,-179.400,6.257,148.955
C05134=1162.535,71.527,-50.930,-179.397,6.258,148.955
C05135=1162.531,71.777,-50.947,-179.395,6.259,148.954
C05136=1162.525,72.026,-50.964,-179.392,6.260,148.953
C05137=1162.520,72.275,-50.980,-179.390,6.261,148.953
C05138=1162.516,72.525,-50.997,-179.387,6.263,148.952
C05139=1162.511,72.774,-51.014,-179.384,6.264,148.952
C05140=1162.506,73.024,-51.031,-179.382,6.265,148.951
C05141=1162.500,73.273,-51.048,-179.379,6.266,148.951
C05142=1162.496,73.522,-51.065,-179.376,6.267,148.950
C05143=1162.491,73.772,-51.082,-179.374,6.268,148.950
C05144=1162.486,74.022,-51.099,-179.371,6.270,148.949
C05145=1162.481,74.270,-51.116,-179.369,6.270,148.949
C05146=1162.476,74.520,-51.133,-179.366,6.272,148.948
C05147=1162.472,74.769,-51.149,-179.363,6.273,148.948
C05148=1162.466,75.019,-51.167,-179.360,6.274,148.947
C05149=1162.461,75.268,-51.183,-179.357,6.276,148.947
C05150=1162.456,75.518,-51.200,-179.355,6.277,148.946
C05151=1162.452,75.767,-51.217,-179.352,6.278,148.946
C05152=1162.447,76.016,-51.235,-179.350,6.279,148.945
C05153=1162.442,76.265,-51.251,-179.347,6.280,148.945
C05154=1162.436,76.515,-51.269,-179.345,6.281,148.944
C05155=1162.432,76.764,-51.285,-179.342,6.283,148.944
C05156=1162.427,77.014,-51.302,-179.339,6.283,148.943
C05157=1162.423,77.263,-51.320,-179.337,6.285,148.943
C05158=1162.417,77.512,-51.337,-179.333,6.286,148.942
C05159=1162.411,77.762,-51.354,-179.331,6.287,148.941
C05160=1162.407,78.011,-51.371,-179.328,6.289,148.941
C05161=1162.402,78.260,-51.389,-179.326,6.289,148.940
C05162=1162.398,78.510,-51.405,-179.323,6.291,148.940
C05163=1162.392,78.760,-51.423,-179.321,6.292,148.940
C05164=1162.388,79.008,-51.440,-179.318,6.293,148.939
C05165=1162.382,79.258,-51.457,-179.315,6.295,148.938
C05166=1162.377,79.507,-51.474,-179.312,6.295,148.938
C05167=1162.373,79.776,-51.492,-179.310,6.297,148.937
C05168=1162.367,80.044,-51.511,-179.306,6.298,148.937
C05169=1162.361,80.312,-51.530,-179.304,6.299,148.936
C05170=1162.357,80.581,-51.548,-179.301,6.301,148.936
C05171=1162.352,80.830,-51.566,-179.298,6.302,148.935
C05172=1162.346,81.079,-51.583,-179.296,6.303,148.935
C05173=1162.342,81.329,-51.600,-179.293,6.304,148.934
C05174=1162.337,81.578,-51.618,-179.290,6.306,148.934
C05175=1162.331,81.828,-51.635,-179.288,6.307,148.933
C05176=1162.327,82.077,-51.652,-179.285,6.308,148.933
C05177=1162.322,82.326,-51.669,-179.283,6.309,148.932
C05178=1162.317,82.576,-51.687,-179.280,6.311,148.932
C05179=1162.313,82.825,-51.704,-179.277,6.312,148.931
C05180=1162.307,83.075,-51.721,-179.274,6.313,148.931
C05181=1162.302,83.323,-51.739,-179.271,6.314,148.930
C05182=1162.297,83.573,-51.756,-179.269,6.315,148.930
C05183=1162.293,83.822,-51.774,-179.266,6.317,148.929
C05184=1162.287,84.072,-51.791,-179.263,6.318,148.929
C05185=1162.282,84.321,-51.809,-179.261,6.319,148.928
C05186=1162.278,84.570,-51.826,-179.258,6.321,148.928
C05187=1162.273,84.820,-51.844,-179.256,6.321,148.927
C05188=1162.268,85.069,-51.861,-179.253,6.323,148.927
C05189=1162.263,85.319,-51.879,-179.250,6.324,148.926
C05190=1162.259,85.567,-51.896,-179.248,6.325,148.926
C05191=1162.254,85.817,-51.913,-179.245,6.327,148.925
C05192=1162.249,86.066,-51.931,-179.242,6.328,148.925
C05193=1162.243,86.316,-51.949,-179.240,6.329,148.924
C05194=1162.238,86.565,-51.967,-179.237,6.331,148.924
C05195=1162.234,86.814,-51.984,-179.234,6.331,148.923
C05196=1162.229,87.064,-52.001,-179.232,6.333,148.923
C05197=1162.224,87.313,-52.019,-179.229,6.335,148.922
C05198=1162.219,87.563,-52.037,-179.226,6.335,148.922
C05199=1162.214,87.812,-52.055,-179.223,6.337,148.921
C05200=1162.209,88.061,-52.073,-179.221,6.338,148.920
C05201=1162.205,88.311,-52.089,-179.218,6.339,148.920
C05202=1162.200,88.560,-52.107,-179.215,6.341,148.920
C05203=1162.195,88.809,-52.125,-179.213,6.341,148.919
C05204=1162.190,89.058,-52.143,-179.210,6.343,148.919
C05205=1162.185,89.308,-52.160,-179.207,6.345,148.918
C05206=1162.180,89.557,-52.178,-179.205,6.345,148.917
C05207=1162.175,89.807,-52.196,-179.202,6.347,148.917
C05208=1162.170,90.056,-52.213,-179.199,6.349,148.917
C05209=1162.165,90.305,-52.231,-179.197,6.349,148.916
C05210=1162.161,90.554,-52.249,-179.194,6.351,148.916
C05211=1162.156,90.804,-52.267,-179.192,6.352,148.915
C05212=1162.151,91.053,-52.285,-179.189,6.354,148.915
C05213=1162.146,91.303,-52.302,-179.186,6.355,148.914
C05214=1162.141,91.552,-52.320,-179.184,6.356,148.914
C05215=1162.136,91.801,-52.338,-179.181,6.358,148.913
C05216=1162.131,92.050,-52.356,-179.178,6.359,148.913
C05217=1162.126,92.299,-52.374,-179.176,6.360,148.912
C05218=1162.121,92.548,-52.392,-179.173,6.361,148.912
C05219=1162.116,92.798,-52.409,-179.170,6.363,148.911
C05220=1162.111,93.048,-52.428,-179.168,6.364,148.911
C05221=1162.107,93.297,-52.446,-179.165,6.365,148.910
C05222=1162.102,93.546,-52.464,-179.162,6.367,148.910
C05223=1162.097,93.796,-52.482,-179.159,6.368,148.909
C05224=1162.092,94.045,-52.500,-179.157,6.369,148.909
C05225=1162.087,94.294,-52.518,-179.154,6.371,148.908
C05226=1162.082,94.543,-52.536,-179.151,6.371,148.908
C05227=1162.077,94.792,-52.554,-179.149,6.373,148.907
C05228=1162.072,95.041,-52.572,-179.145,6.375,148.907
C05229=1162.067,95.291,-52.590,-179.143,6.375,148.906
C05230=1162.063,95.541,-52.607,-179.141,6.377,148.906
C05231=1162.058,95.790,-52.625,-179.138,6.379,148.905
C05232=1162.053,96.040,-52.643,-179.135,6.380,148.905
C05233=1162.048,96.289,-52.661,-179.133,6.381,148.904
C05234=1162.043,96.538,-52.679,-179.130,6.383,148.904
C05235=1162.038,96.787,-52.697,-179.127,6.384,148.903
C05236=1162.033,97.036,-52.716,-179.124,6.385,148.903
C05237=1162.029,97.285,-52.734,-179.122,6.387,148.902
C05238=1162.023,97.535,-52.753,-179.119,6.388,148.902
C05239=1162.019,97.784,-52.771,-179.116,6.389,148.901
C05240=1162.014,98.033,-52.789,-179.114,6.391,148.901
C05241=1162.009,98.282,-52.807,-179.111,6.392,148.901
C05242=1162.004,98.532,-52.825,-179.108,6.393,148.900
C05243=1162.000,98.782,-52.843,-179.106,6.395,148.900
C05244=1161.995,99.031,-52.861,-179.103,6.396,148.899
C05245=1161.990,99.280,-52.879,-179.100,6.398,148.898
C05246=1161.984,99.529,-52.897,-179.098,6.398,148.898
C05247=1161.980,99.779,-52.917,-179.095,6.400,148.898
C05248=1161.975,100.028,-52.935,-179.092,6.402,148.897
C05249=1161.970,100.277,-52.953,-179.089,6.402,148.897
C05250=1161.965,100.526,-52.970,-179.087,6.404,148.896
C05251=1161.960,100.776,-52.989,-179.084,6.406,148.896
C05252=1161.955,101.026,-53.007,-179.081,6.408,148.895
C05253=1161.951,101.274,-53.026,-179.079,6.408,148.895
C05254=1161.946,101.523,-53.044,-179.076,6.410,148.894
C05255=1161.941,101.772,-53.062,-179.073,6.411,148.894
C05256=1161.936,102.023,-53.081,-179.070,6.413,148.893
C05257=1161.931,102.271,-53.100,-179.068,6.414,148.893
C05258=1161.926,102.520,-53.118,-179.065,6.415,148.892
C05259=1161.921,102.770,-53.136,-179.062,6.417,148.892
C05260=1161.916,103.020,-53.155,-179.060,6.418,148.891
C05261=1161.912,103.268,-53.173,-179.057,6.419,148.891
C05262=1161.907,103.517,-53.191,-179.054,6.421,148.891
C05263=1161.903,103.767,-53.210,-179.052,6.423,148.890
C05264=1161.897,104.016,-53.229,-179.049,6.423,148.889
C05265=1161.892,104.265,-53.247,-179.046,6.425,148.889
C05266=1161.887,104.515,-53.265,-179.044,6.427,148.889
C05267=1161.883,104.764,-53.285,-179.041,6.428,148.888
C05268=1161.878,105.013,-53.303,-179.038,6.429,148.888
C05269=1161.873,105.262,-53.320,-179.036,6.431,148.887
C05270=1161.868,105.512,-53.340,-179.033,6.432,148.887
C05271=1161.863,105.780,-53.360,-179.030,6.434,148.886
C05272=1161.857,106.049,-53.380,-179.027,6.435,148.886
C05273=1161.852,106.316,-53.400,-179.024,6.437,148.885
C05274=1161.847,106.586,-53.420,-179.021,6.438,148.885
C05275=1161.842,106.835,-53.438,-179.018,6.440,148.884
C05276=1161.838,107.083,-53.457,-179.016,6.441,148.884
C05277=1161.833,107.334,-53.476,-179.013,6.442,148.883
C05278=1161.828,107.582,-53.494,-179.010,6.444,148.883
C05279=1161.822,107.832,-53.513,-179.007,6.446,148.882
C05280=1161.818,108.081,-53.532,-179.005,6.447,148.882
C05281=1161.813,108.330,-53.550,-179.002,6.448,148.881
C05282=1161.808,108.579,-53.569,-178.999,6.450,148.881
C05283=1161.804,108.829,-53.588,-178.997,6.451,148.881
C05284=1161.798,109.078,-53.607,-178.995,6.452,148.880
C05285=1161.794,109.328,-53.625,-178.991,6.454,148.880
C05286=1161.790,109.576,-53.644,-178.989,6.455,148.879
C05287=1161.784,109.826,-53.663,-178.986,6.457,148.879
C05288=1161.780,110.075,-53.682,-178.983,6.459,148.878
C05289=1161.775,110.324,-53.701,-178.981,6.460,148.878
C05290=1161.770,110.574,-53.719,-178.978,6.461,148.877
C05291=1161.765,110.823,-53.739,-178.975,6.463,148.877
C05292=1161.760,111.072,-53.756,-178.972,6.465,148.876
C05293=1161.755,111.321,-53.776,-178.970,6.466,148.876
C05294=1161.751,111.570,-53.795,-178.967,6.467,148.875
C05295=1161.746,111.820,-53.814,-178.964,6.468,148.875
C05296=1161.741,112.069,-53.832,-178.962,6.470,148.875
C05297=1161.736,112.318,-53.852,-178.959,6.472,148.874
C05298=1161.731,112.567,-53.870,-178.956,6.474,148.874
C05299=1161.726,112.816,-53.889,-178.954,6.474,148.873
C05300=1161.721,113.066,-53.909,-178.951,6.476,148.873
C05301=1161.716,113.315,-53.927,-178.948,6.478,148.872
C05302=1161.712,113.565,-53.947,-178.945,6.479,148.872
C05303=1161.707,113.813,-53.965,-178.943,6.481,148.872
C05304=1161.702,114.063,-53.985,-178.940,6.482,148.871
C05305=1161.697,114.312,-54.003,-178.937,6.483,148.870
C05306=1161.693,114.561,-54.023,-178.935,6.485,148.870
C05307=1161.687,114.810,-54.042,-178.932,6.487,148.870
C05308=1161.683,115.060,-54.061,-178.929,6.488,148.869
C05309=1161.678,115.309,-54.080,-178.926,6.490,148.869
C05310=1161.674,115.558,-54.099,-178.924,6.491,148.868
C05311=1161.668,115.807,-54.118,-178.921,6.492,148.868
C05312=1161.663,116.057,-54.138,-178.919,6.494,148.867
C05313=1161.659,116.305,-54.156,-178.916,6.496,148.867
C05314=1161.654,116.555,-54.176,-178.913,6.497,148.866
C05315=1161.648,116.804,-54.195,-178.910,6.498,148.866
C05316=1161.644,117.054,-54.214,-178.908,6.500,148.866
C05317=1161.639,117.302,-54.233,-178.905,6.501,148.865
C05318=1161.634,117.552,-54.253,-178.902,6.503,148.865
C05319=1161.630,117.801,-54.271,-178.899,6.505,148.864
C05320=1161.625,118.050,-54.291,-178.896,6.506,148.864
C05321=1161.620,118.300,-54.311,-178.894,6.508,148.863
C05322=1161.615,118.549,-54.330,-178.892,6.509,148.863
C05323=1161.611,118.798,-54.349,-178.889,6.511,148.863
C05324=1161.606,119.047,-54.368,-178.886,6.512,148.862
C05325=1161.601,119.296,-54.388,-178.883,6.514,148.862
C05326=1161.596,119.545,-54.407,-178.880,6.515,148.861
C05327=1161.592,119.794,-54.426,-178.878,6.517,148.861
C05328=1161.587,120.044,-54.446,-178.875,6.518,148.860
C05329=1161.581,120.293,-54.465,-178.873,6.520,148.860
C05330=1161.577,120.542,-54.484,-178.869,6.521,148.859
C05331=1161.572,120.791,-54.504,-178.867,6.523,148.859
C05332=1161.567,121.040,-54.523,-178.864,6.524,148.858
C05333=1161.563,121.290,-54.543,-178.861,6.526,148.858
C05334=1161.557,121.539,-54.562,-178.859,6.528,148.858
C05335=1161.553,121.788,-54.581,-178.856,6.530,148.857
C05336=1161.548,122.037,-54.600,-178.854,6.531,148.857
C05337=1161.543,122.287,-54.620,-178.851,6.532,148.856
C05338=1161.538,122.536,-54.640,-178.848,6.534,148.856
C05339=1161.533,122.785,-54.659,-178.845,6.535,148.855
C05340=1161.529,123.034,-54.678,-178.842,6.537,148.855
C05341=1161.525,123.283,-54.699,-178.840,6.539,148.855
C05342=1161.519,123.532,-54.718,-178.837,6.540,148.854
C05343=1161.515,123.782,-54.737,-178.834,6.542,148.854
C05344=1161.510,124.031,-54.757,-178.832,6.543,148.853
C05345=1161.504,124.280,-54.776,-178.829,6.544,148.853
C05346=1161.500,124.530,-54.796,-178.826,6.546,148.852
C05347=1161.495,124.779,-54.816,-178.824,6.548,148.852
C05348=1161.491,125.027,-54.835,-178.821,6.550,148.852
C05349=1161.486,125.277,-54.855,-178.818,6.551,148.851
C05350=1161.481,125.526,-54.874,-178.815,6.553,148.851
C05351=1161.476,125.775,-54.894,-178.812,6.554,148.850
C05352=1161.471,126.024,-54.914,-178.810,6.556,148.850
C05353=1161.467,126.274,-54.934,-178.807,6.557,148.849
C05354=1161.462,126.523,-54.953,-178.805,6.559,148.849
C05355=1161.457,126.772,-54.973,-178.802,6.561,148.849
C05356=1161.452,127.021,-54.993,-178.799,6.562,148.848
C05357=1161.447,127.271,-55.013,-178.797,6.564,148.848
C05358=1161.442,127.519,-55.033,-178.793,6.565,148.847
C05359=1161.438,127.769,-55.052,-178.791,6.567,148.847
C05360=1161.433,128.018,-55.072,-178.788,6.569,148.846
C05361=1161.428,128.267,-55.092,-178.785,6.570,148.846
C05362=1161.423,128.516,-55.112,-178.783,6.572,148.846
C05363=1161.418,128.765,-55.131,-178.780,6.574,148.845
C05364=1161.414,129.014,-55.152,-178.777,6.576,148.845
C05365=1161.409,129.264,-55.171,-178.775,6.577,148.844
C05366=1161.404,129.513,-55.191,-178.772,6.578,148.844
C05367=1161.399,129.762,-55.211,-178.769,6.580,148.843
C05368=1161.395,130.011,-55.231,-178.766,6.581,148.843
C05369=1161.390,130.260,-55.251,-178.764,6.583,148.843
C05370=1161.385,130.510,-55.271,-178.761,6.585,148.842
C05371=1161.380,130.758,-55.291,-178.758,6.587,148.842
C05372=1161.376,131.008,-55.310,-178.756,6.588,148.841
C05373=1161.371,131.257,-55.331,-178.753,6.590,148.841
C05374=1161.366,131.506,-55.350,-178.750,6.592,148.841
C05375=1161.361,131.775,-55.372,-178.747,6.593,148.840
C05376=1161.356,132.043,-55.394,-178.744,6.595,148.840
C05377=1161.351,132.312,-55.416,-178.741,6.597,148.839
C05378=1161.346,132.581,-55.437,-178.738,6.599,148.839
C05379=1161.341,132.830,-55.457,-178.736,6.600,148.838
C05380=1161.336,133.078,-55.477,-178.733,6.601,148.838
C05381=1161.331,133.328,-55.497,-178.730,6.603,148.837
C05382=1161.326,133.577,-55.518,-178.727,6.605,148.837
C05383=1161.322,133.826,-55.537,-178.725,6.607,148.837
C05384=1161.317,134.075,-55.558,-178.722,6.608,148.836
C05385=1161.313,134.324,-55.578,-178.719,6.610,148.836
C05386=1161.307,134.573,-55.597,-178.717,6.612,148.836
C05387=1161.302,134.822,-55.618,-178.714,6.613,148.835
C05388=1161.297,135.072,-55.638,-178.711,6.615,148.835
C05389=1161.293,135.321,-55.658,-178.709,6.617,148.834
C05390=1161.289,135.570,-55.679,-178.706,6.619,148.834
C05391=1161.284,135.819,-55.698,-178.703,6.620,148.834
C05392=1161.279,136.069,-55.719,-178.700,6.622,148.833
C05393=1161.274,136.318,-55.740,-178.697,6.623,148.833
C05394=1161.270,136.567,-55.760,-178.695,6.625,148.832
C05395=1161.264,136.815,-55.779,-178.692,6.627,148.832
C05396=1161.259,137.065,-55.800,-178.689,6.629,148.831
C05397=1161.255,137.314,-55.821,-178.686,6.630,148.831
C05398=1161.250,137.563,-55.841,-178.684,6.632,148.831
C05399=1161.246,137.812,-55.861,-178.681,6.634,148.830
C05400=1161.240,138.061,-55.882,-178.678,6.636,148.830
C05401=1161.236,138.310,-55.902,-178.676,6.637,148.829
C05402=1161.232,138.559,-55.922,-178.673,6.639,148.829
C05403=1161.226,138.809,-55.943,-178.670,6.641,148.829
C05404=1161.222,139.058,-55.963,-178.667,6.642,148.828
C05405=1161.217,139.307,-55.983,-178.665,6.644,148.828
C05406=1161.212,139.556,-56.004,-178.662,6.646,148.827
C05407=1161.208,139.805,-56.025,-178.659,6.648,148.827
C05408=1161.203,140.054,-56.045,-178.657,6.649,148.827
C05409=1161.198,140.304,-56.066,-178.653,6.651,148.826
C05410=1161.193,140.553,-56.086,-178.651,6.652,148.826
C05411=1161.189,140.802,-56.106,-178.648,6.654,148.825
C05412=1161.184,141.051,-56.127,-178.645,6.656,148.825
C05413=1161.179,141.300,-56.148,-178.643,6.658,148.825
C05414=1161.175,141.549,-56.168,-178.640,6.659,148.824
C05415=1161.170,141.799,-56.189,-178.637,6.661,148.824
C05416=1161.165,142.047,-56.209,-178.635,6.663,148.823
C05417=1161.160,142.297,-56.230,-178.632,6.665,148.823
C05418=1161.155,142.546,-56.251,-178.629,6.666,148.823
C05419=1161.151,142.795,-56.271,-178.626,6.668,148.822
C05420=1161.146,143.044,-56.292,-178.624,6.670,148.822
C05421=1161.141,143.293,-56.312,-178.621,6.671,148.821
C05422=1161.136,143.542,-56.333,-178.618,6.673,148.821
C05423=1161.132,143.791,-56.354,-178.616,6.675,148.821
C05424=1161.127,144.040,-56.375,-178.613,6.677,148.820
C05425=1161.122,144.289,-56.395,-178.610,6.678,148.820
C05426=1161.117,144.538,-56.416,-178.607,6.680,148.820
C05427=1161.113,144.787,-56.436,-178.605,6.682,148.819
C05428=1161.107,145.037,-56.457,-178.602,6.684,148.819
C05429=1161.103,145.285,-56.478,-178.599,6.685,148.818
C05430=1161.098,145.534,-56.499,-178.597,6.687,148.818
C05431=1161.094,145.783,-56.520,-178.594,6.689,148.818
C05432=1161.089,146.032,-56.541,-178.591,6.691,148.817
C05433=1161.085,146.282,-56.561,-178.589,6.692,148.817
C05434=1161.080,146.531,-56.582,-178.586,6.694,148.816
C05435=1161.075,146.780,-56.603,-178.583,6.696,148.816
C05436=1161.070,147.029,-56.624,-178.580,6.698,148.816
C05437=1161.066,147.278,-56.645,-178.577,6.700,148.815
C05438=1161.061,147.527,-56.666,-178.574,6.702,148.815
C05439=1161.055,147.776,-56.687,-178.572,6.703,148.815
C05440=1161.051,148.025,-56.707,-178.569,6.705,148.814
C05441=1161.046,148.274,-56.729,-178.566,6.707,148.814
C05442=1161.042,148.524,-56.750,-178.564,6.709,148.813
C05443=1161.037,148.773,-56.770,-178.561,6.710,148.813
C05444=1161.032,149.022,-56.791,-178.558,6.712,148.813
C05445=1161.028,149.271,-56.813,-178.556,6.714,148.812
C05446=1161.023,149.520,-56.833,-178.553,6.716,148.812
C05447=1161.018,149.769,-56.854,-178.550,6.717,148.812
C05448=1161.013,150.017,-56.876,-178.547,6.719,148.811
C05449=1161.009,150.267,-56.897,-178.545,6.721,148.811
C05450=1161.004,150.516,-56.917,-178.542,6.723,148.810
C05451=1160.999,150.765,-56.939,-178.539,6.725,148.810
C05452=1160.994,151.014,-56.960,-178.536,6.727,148.810
C05453=1160.989,151.263,-56.981,-178.533,6.729,148.809
C05454=1160.986,151.512,-57.002,-178.531,6.730,148.809
C05455=1160.980,151.762,-57.023,-178.528,6.732,148.808
C05456=1160.976,152.010,-57.045,-178.525,6.734,148.808
C05457=1160.971,152.259,-57.065,-178.523,6.736,148.808
C05458=1160.966,152.509,-57.086,-178.520,6.738,148.808
C05459=1160.962,152.758,-57.108,-178.518,6.739,148.807
C05460=1160.956,153.007,-57.129,-178.515,6.741,148.807
C05461=1160.952,153.256,-57.150,-178.512,6.743,148.806
C05462=1160.947,153.505,-57.171,-178.510,6.745,148.806
C05463=1160.942,153.753,-57.193,-178.506,6.747,148.806
C05464=1160.938,154.003,-57.214,-178.504,6.749,148.805
C05465=1160.934,154.252,-57.235,-178.501,6.751,148.805
C05466=1160.928,154.501,-57.256,-178.498,6.752,148.805
C05467=1160.924,154.750,-57.278,-178.495,6.754,148.804
C05468=1160.919,155.000,-57.299,-178.493,6.756,148.804
C05469=1160.914,155.248,-57.321,-178.490,6.758,148.803
C05470=1160.910,155.497,-57.342,-178.487,6.759,148.803
C05471=1160.905,155.746,-57.363,-178.485,6.761,148.803
C05472=1160.901,155.995,-57.385,-178.481,6.764,148.802
C05473=1160.895,156.244,-57.406,-178.479,6.765,148.802
C05474=1160.890,156.493,-57.428,-178.476,6.767,148.802
C05475=1160.886,156.743,-57.449,-178.474,6.769,148.801
C05476=1160.882,156.991,-57.470,-178.471,6.771,148.801
C05477=1160.877,157.240,-57.492,-178.468,6.773,148.801
C05478=1160.872,157.490,-57.513,-178.466,6.774,148.800
C05479=1160.867,157.758,-57.537,-178.462,6.777,148.800
C05480=1160.862,158.027,-57.560,-178.460,6.779,148.800
C05481=1160.856,158.296,-57.583,-178.457,6.780,148.799
C05482=1160.852,158.565,-57.607,-178.453,6.783,148.799
C05483=1160.847,158.815,-57.628,-178.451,6.785,148.798
C05484=1160.842,159.063,-57.650,-178.448,6.786,148.798
C05485=1160.838,159.312,-57.671,-178.446,6.788,148.798
C05486=1160.833,159.562,-57.693,-178.443,6.790,148.797
C05487=1160.828,159.811,-57.714,-178.440,6.793,148.797
C05488=1160.823,160.059,-57.736,-178.437,6.794,148.797
C05489=1160.819,160.309,-57.758,-178.434,6.796,148.796
C05490=1160.814,160.557,-57.780,-178.432,6.798,148.796
C05491=1160.809,160.807,-57.801,-178.429,6.799,148.795
C05492=1160.805,161.056,-57.823,-178.426,6.801,148.795
C05493=1160.800,161.305,-57.844,-178.424,6.803,148.795
C05494=1160.796,161.554,-57.867,-178.421,6.806,148.795
C05495=1160.791,161.803,-57.888,-178.418,6.808,148.794
C05496=1160.786,162.051,-57.910,-178.415,6.809,148.794
